C03657=1167.639,225.132,-63.200,-177.659,7.224,148.674
C03658=1167.644,224.883,-63.174,-177.662,7.221,148.674
C03659=1167.648,224.634,-63.149,-177.665,7.219,148.674
C03660=1167.653,224.386,-63.123,-177.668,7.216,148.674
C03661=1167.657,224.138,-63.098,-177.670,7.214,148.674
C03662=1167.661,223.888,-63.073,-177.673,7.212,148.675
C03663=1167.666,223.640,-63.047,-177.676,7.210,148.675
C03664=1167.670,223.391,-63.021,-177.679,7.207,148.675
C03665=1167.675,223.142,-62.996,-177.681,7.205,148.675
C03666=1167.680,222.894,-62.970,-177.684,7.202,148.675
C03667=1167.684,222.645,-62.945,-177.686,7.200,148.676
C03668=1167.689,222.397,-62.920,-177.689,7.197,148.676
C03669=1167.693,222.148,-62.894,-177.692,7.195,148.676
C03670=1167.698,221.899,-62.869,-177.695,7.192,148.676
C03671=1167.702,221.650,-62.844,-177.697,7.191,148.676
C03672=1167.707,221.402,-62.818,-177.700,7.188,148.677
C03673=1167.712,221.153,-62.793,-177.703,7.186,148.677
C03674=1167.715,220.904,-62.768,-177.705,7.183,148.677
C03675=1167.720,220.656,-62.743,-177.708,7.181,148.677
C03676=1167.725,220.407,-62.718,-177.711,7.178,148.677
C03677=1167.729,220.158,-62.692,-177.714,7.176,148.678
C03678=1167.734,219.910,-62.667,-177.716,7.174,148.678
C03679=1167.738,219.661,-62.642,-177.719,7.171,148.678
C03680=1167.742,219.413,-62.617,-177.722,7.169,148.678
C03681=1167.747,219.163,-62.592,-177.724,7.166,148.678
C03682=1167.752,218.915,-62.566,-177.727,7.164,148.679
C03683=1167.756,218.666,-62.541,-177.730,7.161,148.679
C03684=1167.761,218.418,-62.516,-177.733,7.159,148.679
C03685=1167.765,218.169,-62.491,-177.735,7.157,148.679
C03686=1167.770,217.921,-62.466,-177.738,7.155,148.679
C03687=1167.774,217.671,-62.441,-177.740,7.152,148.680
C03688=1167.779,217.423,-62.416,-177.743,7.150,148.680
C03689=1167.783,217.174,-62.391,-177.746,7.148,148.680
C03690=1167.788,216.926,-62.366,-177.749,7.145,148.680
C03691=1167.792,216.676,-62.341,-177.751,7.143,148.680
C03692=1167.797,216.428,-62.315,-177.754,7.140,148.681
C03693=1167.801,216.179,-62.291,-177.757,7.138,148.681
C03694=1167.806,215.931,-62.266,-177.760,7.136,148.681
C03695=1167.810,215.682,-62.241,-177.762,7.134,148.681
C03696=1167.815,215.433,-62.216,-177.765,7.131,148.682
C03697=1167.819,215.184,-62.191,-177.767,7.129,148.682
C03698=1167.824,214.936,-62.166,-177.771,7.126,148.682
C03699=1167.829,214.687,-62.141,-177.773,7.124,148.682
C03700=1167.833,214.438,-62.116,-177.776,7.122,148.682
C03701=1167.838,214.190,-62.092,-177.779,7.120,148.683
C03702=1167.842,213.940,-62.067,-177.781,7.117,148.683
C03703=1167.846,213.693,-62.042,-177.784,7.115,148.683
C03704=1167.851,213.443,-62.017,-177.786,7.113,148.683
C03705=1167.855,213.195,-61.993,-177.790,7.110,148.684
C03706=1167.860,212.946,-61.968,-177.792,7.108,148.684
C03707=1167.865,212.697,-61.942,-177.795,7.106,148.684
C03708=1167.869,212.449,-61.918,-177.797,7.103,148.684
C03709=1167.873,212.199,-61.893,-177.800,7.101,148.685
C03710=1167.878,211.951,-61.869,-177.803,7.099,148.685
C03711=1167.883,211.703,-61.844,-177.806,7.096,148.685
C03712=1167.887,211.453,-61.819,-177.809,7.094,148.685
C03713=1167.892,211.205,-61.795,-177.811,7.092,148.685
C03714=1167.897,210.956,-61.770,-177.814,7.090,148.686
C03715=1167.901,210.707,-61.745,-177.816,7.087,148.686
C03716=1167.906,210.437,-61.719,-177.819,7.085,148.686
C03717=1167.910,210.166,-61.692,-177.823,7.082,148.687
C03718=1167.915,209.896,-61.665,-177.825,7.080,148.687
C03719=1167.921,209.626,-61.638,-177.828,7.078,148.687
C03720=1167.925,209.376,-61.613,-177.831,7.075,148.687
C03721=1167.929,209.128,-61.589,-177.834,7.073,148.687
C03722=1167.935,208.879,-61.564,-177.836,7.071,148.688
C03723=1167.938,208.630,-61.540,-177.839,7.068,148.688
C03724=1167.944,208.381,-61.515,-177.842,7.066,148.688
C03725=1167.948,208.133,-61.491,-177.844,7.063,148.688
C03726=1167.953,207.884,-61.467,-177.847,7.062,148.689
C03727=1167.957,207.635,-61.442,-177.850,7.059,148.689
C03728=1167.961,207.387,-61.418,-177.853,7.057,148.689
C03729=1167.966,207.138,-61.393,-177.855,7.055,148.689
C03730=1167.970,206.889,-61.369,-177.858,7.052,148.689
C03731=1167.975,206.640,-61.344,-177.861,7.050,148.690
C03732=1167.980,206.392,-61.320,-177.864,7.048,148.690
C03733=1167.985,206.143,-61.296,-177.866,7.046,148.690
C03734=1167.989,205.894,-61.271,-177.869,7.044,148.691
C03735=1167.993,205.645,-61.247,-177.872,7.041,148.691
C03736=1167.998,205.397,-61.222,-177.874,7.039,148.691
C03737=1168.003,205.148,-61.199,-177.877,7.036,148.691
C03738=1168.007,204.899,-61.175,-177.880,7.034,148.691
C03739=1168.012,204.650,-61.150,-177.882,7.033,148.692
C03740=1168.016,204.401,-61.126,-177.885,7.030,148.692
C03741=1168.021,204.153,-61.102,-177.888,7.028,148.692
C03742=1168.025,203.904,-61.077,-177.891,7.025,148.693
C03743=1168.030,203.655,-61.053,-177.893,7.023,148.693
C03744=1168.034,203.406,-61.029,-177.896,7.021,148.693
C03745=1168.039,203.157,-61.005,-177.899,7.019,148.693
C03746=1168.044,202.909,-60.981,-177.901,7.017,148.694
C03747=1168.048,202.660,-60.956,-177.904,7.015,148.694
C03748=1168.053,202.411,-60.932,-177.907,7.012,148.694
C03749=1168.057,202.162,-60.908,-177.909,7.010,148.694
C03750=1168.062,201.914,-60.884,-177.913,7.008,148.695
C03751=1168.066,201.665,-60.861,-177.915,7.006,148.695
C03752=1168.071,201.415,-60.836,-177.918,7.004,148.695
C03753=1168.075,201.167,-60.812,-177.920,7.001,148.695
C03754=1168.080,200.918,-60.787,-177.923,6.999,148.696
C03755=1168.084,200.669,-60.764,-177.926,6.997,148.696
C03756=1168.089,200.421,-60.740,-177.928,6.994,148.696
C03757=1168.094,200.172,-60.716,-177.931,6.993,148.696
C03758=1168.098,199.923,-60.692,-177.934,6.991,148.697
C03759=1168.102,199.674,-60.668,-177.937,6.988,148.697
C03760=1168.107,199.425,-60.644,-177.939,6.986,148.697
C03761=1168.112,199.177,-60.620,-177.943,6.983,148.697
C03762=1168.117,198.927,-60.596,-177.945,6.981,148.698
C03763=1168.121,198.679,-60.572,-177.947,6.980,148.698
C03764=1168.126,198.431,-60.548,-177.951,6.977,148.698
C03765=1168.130,198.182,-60.525,-177.953,6.975,148.698
C03766=1168.134,197.932,-60.500,-177.956,6.973,148.699
C03767=1168.139,197.683,-60.477,-177.959,6.971,148.699
C03768=1168.143,197.435,-60.453,-177.961,6.968,148.699
C03769=1168.148,197.186,-60.429,-177.964,6.967,148.700
C03770=1168.153,196.937,-60.405,-177.967,6.964,148.700
C03771=1168.158,196.688,-60.381,-177.969,6.962,148.700
C03772=1168.162,196.440,-60.357,-177.972,6.960,148.700
C03773=1168.167,196.191,-60.334,-177.975,6.958,148.701
C03774=1168.171,195.942,-60.310,-177.977,6.955,148.701
C03775=1168.176,195.693,-60.287,-177.980,6.954,148.701
C03776=1168.181,195.444,-60.263,-177.983,6.951,148.701
C03777=1168.185,195.196,-60.239,-177.985,6.949,148.702
C03778=1168.190,194.947,-60.216,-177.988,6.947,148.702
C03779=1168.195,194.698,-60.192,-177.991,6.945,148.702
C03780=1168.199,194.449,-60.168,-177.993,6.942,148.702
C03781=1168.204,194.200,-60.145,-177.996,6.941,148.703
C03782=1168.207,193.951,-60.120,-177.999,6.939,148.703
C03783=1168.212,193.702,-60.097,-178.002,6.936,148.703
C03784=1168.217,193.453,-60.074,-178.004,6.934,148.704
C03785=1168.222,193.204,-60.050,-178.007,6.932,148.704
C03786=1168.226,192.956,-60.026,-178.010,6.930,148.704
C03787=1168.231,192.707,-60.003,-178.012,6.928,148.704
C03788=1168.235,192.458,-59.980,-178.015,6.926,148.705
C03789=1168.240,192.209,-59.956,-178.018,6.923,148.705
C03790=1168.244,191.960,-59.932,-178.021,6.921,148.705
C03791=1168.250,191.712,-59.909,-178.023,6.919,148.706
C03792=1168.254,191.463,-59.886,-178.026,6.917,148.706
C03793=1168.259,191.214,-59.862,-178.029,6.915,148.706
C03794=1168.264,190.965,-59.838,-178.031,6.913,148.706
C03795=1168.268,190.716,-59.815,-178.034,6.911,148.707
C03796=1168.273,190.467,-59.792,-178.037,6.909,148.707
C03797=1168.277,190.219,-59.769,-178.039,6.907,148.707
C03798=1168.282,189.970,-59.746,-178.042,6.905,148.708
C03799=1168.286,189.721,-59.722,-178.045,6.902,148.708
C03800=1168.291,189.472,-59.698,-178.048,6.900,148.708
C03801=1168.295,189.223,-59.675,-178.050,6.898,148.708
C03802=1168.300,188.974,-59.651,-178.053,6.897,148.709
C03803=1168.305,188.725,-59.628,-178.056,6.894,148.709
C03804=1168.309,188.476,-59.605,-178.059,6.892,148.709
C03805=1168.313,188.227,-59.582,-178.061,6.890,148.710
C03806=1168.319,187.979,-59.559,-178.064,6.888,148.710
C03807=1168.323,187.730,-59.536,-178.067,6.886,148.710
C03808=1168.328,187.481,-59.512,-178.070,6.884,148.711
C03809=1168.333,187.232,-59.489,-178.072,6.882,148.711
C03810=1168.337,186.983,-59.466,-178.075,6.879,148.711
C03811=1168.342,186.734,-59.443,-178.078,6.877,148.711
C03812=1168.346,186.485,-59.419,-178.081,6.876,148.712
C03813=1168.351,186.236,-59.396,-178.083,6.874,148.712
C03814=1168.355,185.987,-59.373,-178.086,6.871,148.712
C03815=1168.360,185.739,-59.350,-178.089,6.869,148.713
C03816=1168.365,185.490,-59.327,-178.091,6.867,148.713
C03817=1168.370,185.241,-59.304,-178.094,6.865,148.713
C03818=1168.374,184.992,-59.281,-178.097,6.863,148.713
C03819=1168.378,184.743,-59.257,-178.100,6.861,148.714
C03820=1168.384,184.473,-59.232,-178.102,6.859,148.714
C03821=1168.388,184.204,-59.208,-178.105,6.857,148.715
C03822=1168.393,183.934,-59.183,-178.108,6.855,148.715
C03823=1168.399,183.664,-59.158,-178.111,6.852,148.715
C03824=1168.403,183.416,-59.135,-178.114,6.850,148.715
C03825=1168.407,183.167,-59.112,-178.116,6.848,148.716
C03826=1168.413,182.918,-59.089,-178.120,6.846,148.716
C03827=1168.417,182.670,-59.066,-178.122,6.844,148.716
C03828=1168.422,182.420,-59.043,-178.125,6.842,148.717
C03829=1168.426,182.171,-59.020,-178.127,6.840,148.717
C03830=1168.430,181.922,-58.997,-178.130,6.838,148.717
C03831=1168.436,181.674,-58.974,-178.133,6.836,148.718
C03832=1168.440,181.425,-58.951,-178.136,6.834,148.718
C03833=1168.445,181.175,-58.929,-178.138,6.832,148.718
C03834=1168.449,180.926,-58.905,-178.141,6.830,148.718
C03835=1168.454,180.678,-58.883,-178.144,6.828,148.719
C03836=1168.459,180.429,-58.860,-178.147,6.826,148.719
C03837=1168.463,180.180,-58.838,-178.149,6.824,148.720
C03838=1168.468,179.931,-58.814,-178.152,6.822,148.720
C03839=1168.472,179.682,-58.793,-178.154,6.820,148.720
C03840=1168.477,179.433,-58.769,-178.157,6.818,148.720
C03841=1168.482,179.184,-58.746,-178.160,6.816,148.721
C03842=1168.486,178.935,-58.724,-178.163,6.814,148.721
C03843=1168.491,178.687,-58.701,-178.165,6.812,148.721
C03844=1168.495,178.438,-58.678,-178.168,6.810,148.722
C03845=1168.500,178.188,-58.655,-178.171,6.808,148.722
C03846=1168.504,177.940,-58.633,-178.174,6.806,148.722
C03847=1168.510,177.691,-58.610,-178.176,6.804,148.723
C03848=1168.514,177.442,-58.588,-178.179,6.802,148.723
C03849=1168.519,177.192,-58.565,-178.182,6.801,148.723
C03850=1168.524,176.944,-58.543,-178.184,6.798,148.723
C03851=1168.527,176.695,-58.520,-178.187,6.796,148.724
C03852=1168.532,176.446,-58.497,-178.190,6.794,148.724
C03853=1168.537,176.198,-58.475,-178.192,6.792,148.725
C03854=1168.542,175.948,-58.452,-178.195,6.791,148.725
C03855=1168.546,175.699,-58.429,-178.198,6.788,148.725
C03856=1168.552,175.450,-58.407,-178.201,6.786,148.725
C03857=1168.556,175.201,-58.385,-178.203,6.784,148.726
C03858=1168.561,174.952,-58.362,-178.206,6.782,148.726
C03859=1168.565,174.703,-58.340,-178.209,6.781,148.727
C03860=1168.569,174.455,-58.317,-178.211,6.779,148.727
C03861=1168.574,174.205,-58.295,-178.215,6.776,148.727
C03862=1168.579,173.957,-58.272,-178.217,6.774,148.727
C03863=1168.583,173.708,-58.250,-178.219,6.772,148.728
C03864=1168.589,173.459,-58.228,-178.222,6.771,148.728
C03865=1168.593,173.210,-58.205,-178.225,6.769,148.728
C03866=1168.598,172.960,-58.182,-178.228,6.767,148.729
C03867=1168.603,172.712,-58.161,-178.231,6.765,148.729
C03868=1168.607,172.463,-58.138,-178.233,6.763,148.730
C03869=1168.612,172.214,-58.116,-178.236,6.761,148.730
C03870=1168.617,171.965,-58.094,-178.238,6.759,148.730
C03871=1168.620,171.716,-58.071,-178.241,6.757,148.730
C03872=1168.625,171.467,-58.049,-178.244,6.755,148.731
C03873=1168.630,171.218,-58.027,-178.247,6.753,148.731
C03874=1168.635,170.970,-58.004,-178.250,6.751,148.731
C03875=1168.639,170.720,-57.982,-178.252,6.749,148.732
C03876=1168.645,170.471,-57.960,-178.255,6.748,148.732
C03877=1168.649,170.222,-57.938,-178.258,6.746,148.733
C03878=1168.653,169.973,-57.916,-178.260,6.744,148.733
C03879=1168.658,169.725,-57.893,-178.263,6.742,148.733
C03880=1168.663,169.475,-57.871,-178.266,6.739,148.733
C03881=1168.668,169.226,-57.849,-178.269,6.738,148.734
C03882=1168.672,168.977,-57.827,-178.271,6.736,148.734
C03883=1168.677,168.728,-57.805,-178.274,6.734,148.735
C03884=1168.682,168.479,-57.782,-178.277,6.732,148.735
C03885=1168.686,168.231,-57.760,-178.279,6.731,148.735
C03886=1168.691,167.981,-57.738,-178.282,6.729,148.736
C03887=1168.696,167.733,-57.717,-178.284,6.727,148.736
C03888=1168.700,167.483,-57.695,-178.288,6.724,148.736
C03889=1168.705,167.235,-57.672,-178.290,6.722,148.737
C03890=1168.710,166.985,-57.650,-178.293,6.721,148.737
C03891=1168.715,166.737,-57.629,-178.296,6.719,148.737
C03892=1168.719,166.487,-57.606,-178.298,6.717,148.738
C03893=1168.724,166.239,-57.585,-178.301,6.715,148.738
C03894=1168.728,165.989,-57.563,-178.304,6.714,148.738
C03895=1168.733,165.741,-57.541,-178.306,6.712,148.739
C03896=1168.738,165.491,-57.518,-178.309,6.710,148.739
C03897=1168.743,165.242,-57.497,-178.312,6.708,148.739
C03898=1168.747,164.993,-57.475,-178.315,6.705,148.740
C03899=1168.752,164.744,-57.453,-178.317,6.704,148.740
C03900=1168.757,164.496,-57.431,-178.320,6.702,148.740
C03901=1168.761,164.246,-57.409,-178.323,6.700,148.741
C03902=1168.766,163.998,-57.388,-178.325,6.698,148.741
C03903=1168.770,163.748,-57.366,-178.328,6.697,148.741
C03904=1168.775,163.500,-57.344,-178.331,6.695,148.742
C03905=1168.779,163.250,-57.322,-178.333,6.693,148.742
C03906=1168.784,163.002,-57.300,-178.336,6.691,148.743
C03907=1168.789,162.753,-57.278,-178.339,6.689,148.743
C03908=1168.793,162.504,-57.256,-178.342,6.687,148.743
C03909=1168.798,162.255,-57.235,-178.345,6.685,148.744
C03910=1168.803,162.005,-57.213,-178.347,6.684,148.744
C03911=1168.808,161.756,-57.192,-178.350,6.682,148.744
C03912=1168.813,161.508,-57.170,-178.353,6.680,148.745
C03913=1168.817,161.259,-57.148,-178.355,6.678,148.745
C03914=1168.822,161.010,-57.126,-178.358,6.676,148.745
C03915=1168.826,160.761,-57.104,-178.360,6.674,148.746
C03916=1168.831,160.511,-57.083,-178.363,6.673,148.746
C03917=1168.836,160.263,-57.062,-178.366,6.671,148.746
C03918=1168.840,160.013,-57.040,-178.368,6.669,148.747
C03919=1168.845,159.765,-57.018,-178.371,6.667,148.747
C03920=1168.850,159.515,-56.997,-178.374,6.665,148.748
C03921=1168.855,159.266,-56.975,-178.377,6.663,148.748
C03922=1168.859,159.017,-56.953,-178.380,6.661,148.748
C03923=1168.864,158.769,-56.931,-178.382,6.660,148.749
C03924=1168.869,158.500,-56.909,-178.385,6.658,148.749
C03925=1168.875,158.230,-56.885,-178.388,6.656,148.749
C03926=1168.879,157.961,-56.863,-178.391,6.654,148.750
C03927=1168.884,157.693,-56.839,-178.394,6.652,148.750
C03928=1168.890,157.443,-56.818,-178.397,6.650,148.751
C03929=1168.893,157.194,-56.796,-178.399,6.648,148.751
C03930=1168.898,156.946,-56.774,-178.402,6.647,148.751
C03931=1168.903,156.696,-56.753,-178.405,6.645,148.752
C03932=1168.907,156.447,-56.731,-178.407,6.643,148.752
C03933=1168.913,156.198,-56.710,-178.410,6.641,148.752
C03934=1168.917,155.949,-56.689,-178.413,6.640,148.753
C03935=1168.922,155.701,-56.667,-178.415,6.638,148.753
C03936=1168.926,155.451,-56.646,-178.418,6.636,148.754
C03937=1168.931,155.202,-56.625,-178.421,6.634,148.754
C03938=1168.936,154.953,-56.604,-178.423,6.633,148.754
C03939=1168.941,154.704,-56.582,-178.426,6.631,148.755
C03940=1168.946,154.454,-56.561,-178.429,6.629,148.755
C03941=1168.950,154.206,-56.540,-178.432,6.627,148.755
C03942=1168.955,153.957,-56.519,-178.434,6.626,148.756
C03943=1168.960,153.708,-56.497,-178.437,6.624,148.756
C03944=1168.964,153.458,-56.476,-178.440,6.621,148.757
C03945=1168.969,153.210,-56.455,-178.443,6.620,148.757
C03946=1168.974,152.961,-56.434,-178.446,6.618,148.757
C03947=1168.979,152.712,-56.412,-178.448,6.616,148.758
C03948=1168.984,152.463,-56.391,-178.451,6.614,148.758
C03949=1168.988,152.213,-56.370,-178.454,6.613,148.758
C03950=1168.992,151.964,-56.348,-178.456,6.611,148.759
C03951=1168.998,151.715,-56.328,-178.459,6.609,148.759
C03952=1169.002,151.467,-56.306,-178.462,6.607,148.760
C03953=1169.007,151.218,-56.285,-178.464,6.606,148.760
C03954=1169.012,150.968,-56.264,-178.467,6.604,148.760
C03955=1169.016,150.719,-56.243,-178.470,6.602,148.761
C03956=1169.021,150.470,-56.222,-178.473,6.601,148.761
C03957=1169.026,150.221,-56.201,-178.476,6.599,148.762
C03958=1169.030,149.972,-56.180,-178.478,6.597,148.762
C03959=1169.035,149.723,-56.159,-178.481,6.595,148.762
C03960=1169.040,149.473,-56.138,-178.484,6.594,148.763
C03961=1169.044,149.225,-56.117,-178.486,6.592,148.763
C03962=1169.049,148.976,-56.096,-178.489,6.590,148.764
C03963=1169.054,148.726,-56.075,-178.492,6.588,148.764
C03964=1169.059,148.477,-56.054,-178.495,6.587,148.764
C03965=1169.064,148.229,-56.033,-178.497,6.585,148.765
C03966=1169.068,147.980,-56.012,-178.500,6.583,148.765
C03967=1169.073,147.731,-55.991,-178.503,6.581,148.766
C03968=1169.077,147.481,-55.971,-178.505,6.580,148.766
C03969=1169.082,147.232,-55.950,-178.507,6.579,148.766
C03970=1169.087,146.983,-55.928,-178.510,6.577,148.767
C03971=1169.092,146.734,-55.908,-178.513,6.575,148.767
C03972=1169.097,146.485,-55.887,-178.516,6.574,148.767
C03973=1169.101,146.236,-55.866,-178.518,6.572,148.768
C03974=1169.106,145.987,-55.845,-178.521,6.570,148.768
C03975=1169.111,145.738,-55.825,-178.524,6.568,148.769
C03976=1169.116,145.488,-55.804,-178.526,6.567,148.769
C03977=1169.120,145.240,-55.783,-178.529,6.565,148.769
C03978=1169.125,144.991,-55.762,-178.532,6.563,148.770
C03979=1169.129,144.741,-55.741,-178.535,6.562,148.770
C03980=1169.134,144.492,-55.720,-178.538,6.560,148.771
C03981=1169.139,144.243,-55.700,-178.540,6.558,148.771
C03982=1169.144,143.994,-55.679,-178.543,6.556,148.772
C03983=1169.148,143.745,-55.658,-178.546,6.555,148.772
C03984=1169.154,143.495,-55.637,-178.548,6.553,148.772
C03985=1169.158,143.246,-55.617,-178.551,6.551,148.773
C03986=1169.162,142.998,-55.597,-178.554,6.550,148.773
C03987=1169.168,142.748,-55.576,-178.557,6.548,148.773
C03988=1169.172,142.499,-55.555,-178.559,6.546,148.774
C03989=1169.177,142.250,-55.534,-178.562,6.544,148.774
C03990=1169.182,142.001,-55.514,-178.565,6.543,148.775
C03991=1169.187,141.752,-55.493,-178.567,6.541,148.775
C03992=1169.191,141.503,-55.473,-178.569,6.540,148.775
C03993=1169.196,141.254,-55.452,-178.573,6.538,148.776
C03994=1169.201,141.005,-55.431,-178.575,6.537,148.776
C03995=1169.205,140.756,-55.411,-178.578,6.535,148.777
C03996=1169.210,140.507,-55.391,-178.581,6.533,148.777
C03997=1169.215,140.257,-55.370,-178.583,6.532,148.778
C03998=1169.220,140.008,-55.350,-178.586,6.530,148.778
C03999=1169.224,139.759,-55.330,-178.589,6.528,148.778
C04000=1169.229,139.510,-55.309,-178.592,6.526,148.779
C04001=1169.234,139.261,-55.288,-178.594,6.525,148.779
C04002=1169.238,139.012,-55.268,-178.597,6.523,148.779
C04003=1169.243,138.763,-55.247,-178.600,6.521,148.780
C04004=1169.248,138.513,-55.227,-178.603,6.520,148.780
C04005=1169.253,138.264,-55.207,-178.605,6.519,148.781
C04006=1169.258,138.015,-55.186,-178.608,6.517,148.781
C04007=1169.263,137.767,-55.166,-178.610,6.515,148.782
C04008=1169.267,137.518,-55.146,-178.613,6.514,148.782
C04009=1169.272,137.268,-55.126,-178.616,6.512,148.782
C04010=1169.277,137.019,-55.105,-178.618,6.510,148.783
C04011=1169.282,136.770,-55.085,-178.621,6.508,148.783
C04012=1169.286,136.520,-55.065,-178.624,6.507,148.784
C04013=1169.291,136.271,-55.045,-178.627,6.505,148.784
C04014=1169.296,136.022,-55.024,-178.630,6.504,148.785
C04015=1169.300,135.773,-55.003,-178.632,6.502,148.785
C04016=1169.305,135.524,-54.984,-178.635,6.501,148.785
C04017=1169.309,135.275,-54.963,-178.637,6.499,148.786
C04018=1169.315,135.026,-54.943,-178.640,6.497,148.786
C04019=1169.320,134.776,-54.923,-178.643,6.496,148.787
C04020=1169.324,134.528,-54.903,-178.645,6.494,148.787
C04021=1169.329,134.279,-54.882,-178.649,6.493,148.788
C04022=1169.334,134.029,-54.863,-178.651,6.491,148.788
C04023=1169.338,133.780,-54.842,-178.654,6.489,148.788
C04024=1169.344,133.530,-54.822,-178.657,6.487,148.789
C04025=1169.349,133.282,-54.802,-178.659,6.486,148.789
C04026=1169.353,133.033,-54.782,-178.661,6.485,148.790
C04027=1169.358,132.783,-54.762,-178.664,6.483,148.790
C04028=1169.363,132.514,-54.740,-178.667,6.482,148.791
C04029=1169.368,132.246,-54.718,-178.670,6.480,148.791
C04030=1169.373,131.978,-54.697,-178.673,6.478,148.791
C04031=1169.379,131.709,-54.676,-178.677,6.476,148.792
C04032=1169.383,131.460,-54.655,-178.679,6.475,148.792
C04033=1169.388,131.210,-54.636,-178.681,6.473,148.793
C04034=1169.392,130.961,-54.615,-178.684,6.472,148.793
C04035=1169.398,130.712,-54.596,-178.687,6.470,148.793
C04036=1169.402,130.464,-54.576,-178.689,6.468,148.794
C04037=1169.407,130.214,-54.556,-178.693,6.467,148.794
C04038=1169.412,129.965,-54.535,-178.695,6.465,148.795
C04039=1169.417,129.716,-54.516,-178.698,6.464,148.795
C04040=1169.422,129.467,-54.495,-178.700,6.462,148.796
C04041=1169.426,129.217,-54.476,-178.703,6.461,148.796
C04042=1169.431,128.968,-54.456,-178.706,6.459,148.796
C04043=1169.436,128.720,-54.436,-178.709,6.457,148.797
C04044=1169.441,128.470,-54.416,-178.712,6.456,148.797
C04045=1169.445,128.221,-54.396,-178.714,6.455,148.798
C04046=1169.450,127.971,-54.376,-178.716,6.453,148.798
C04047=1169.455,127.722,-54.357,-178.719,6.451,148.799
C04048=1169.460,127.474,-54.337,-178.722,6.450,148.799
C04049=1169.465,127.224,-54.317,-178.725,6.448,148.800
C04050=1169.469,126.974,-54.297,-178.728,6.446,148.800
C04051=1169.474,126.726,-54.277,-178.730,6.445,148.800
C04052=1169.478,126.477,-54.258,-178.732,6.444,148.801
C04053=1169.483,126.227,-54.239,-178.735,6.442,148.801
C04054=1169.488,125.978,-54.219,-178.738,6.440,148.802
C04055=1169.493,125.730,-54.199,-178.741,6.439,148.802
C04056=1169.498,125.480,-54.179,-178.744,6.437,148.803
C04057=1169.502,125.230,-54.160,-178.746,6.436,148.803
C04058=1169.508,124.982,-54.140,-178.749,6.435,148.804
C04059=1169.512,124.733,-54.120,-178.751,6.433,148.804
C04060=1169.517,124.483,-54.100,-178.755,6.432,148.805
C04061=1169.522,124.234,-54.081,-178.757,6.430,148.805
C04062=1169.527,123.985,-54.061,-178.760,6.428,148.805
C04063=1169.531,123.735,-54.042,-178.762,6.427,148.806
C04064=1169.536,123.487,-54.022,-178.765,6.425,148.806
C04065=1169.541,123.238,-54.003,-178.768,6.424,148.807
C04066=1169.546,122.988,-53.983,-178.771,6.422,148.807
C04067=1169.551,122.739,-53.964,-178.773,6.421,148.808
C04068=1169.556,122.490,-53.944,-178.776,6.420,148.808
C04069=1169.560,122.240,-53.924,-178.778,6.418,148.808
C04070=1169.565,121.991,-53.906,-178.781,6.417,148.809
C04071=1169.569,121.742,-53.885,-178.784,6.415,148.809
C04072=1169.574,121.493,-53.866,-178.787,6.413,148.810
C04073=1169.580,121.244,-53.846,-178.789,6.412,148.810
C04074=1169.584,120.994,-53.827,-178.792,6.410,148.811
C04075=1169.589,120.746,-53.808,-178.795,6.409,148.811
C04076=1169.594,120.496,-53.788,-178.798,6.407,148.812
C04077=1169.598,120.247,-53.769,-178.800,6.406,148.812
C04078=1169.604,119.998,-53.749,-178.802,6.405,148.812
C04079=1169.608,119.749,-53.730,-178.806,6.403,148.813
C04080=1169.613,119.500,-53.711,-178.808,6.402,148.813
C04081=1169.618,119.250,-53.691,-178.811,6.400,148.814
C04082=1169.623,119.001,-53.672,-178.813,6.399,148.814
C04083=1169.627,118.752,-53.653,-178.816,6.397,148.815
C04084=1169.632,118.503,-53.633,-178.819,6.396,148.815
C04085=1169.637,118.254,-53.614,-178.822,6.394,148.816
C04086=1169.642,118.004,-53.594,-178.824,6.392,148.816
C04087=1169.647,117.756,-53.576,-178.827,6.392,148.816
C04088=1169.652,117.505,-53.557,-178.830,6.390,148.817
C04089=1169.656,117.256,-53.537,-178.833,6.388,148.818
C04090=1169.661,117.007,-53.518,-178.835,6.387,148.818
C04091=1169.666,116.758,-53.499,-178.837,6.386,148.818
C04092=1169.671,116.509,-53.479,-178.841,6.384,148.819
C04093=1169.675,116.260,-53.460,-178.843,6.383,148.819
C04094=1169.680,116.011,-53.441,-178.846,6.381,148.820
C04095=1169.685,115.761,-53.421,-178.848,6.380,148.820
C04096=1169.690,115.512,-53.403,-178.851,6.378,148.821
C04097=1169.695,115.262,-53.384,-178.854,6.377,148.821
C04098=1169.700,115.013,-53.365,-178.857,6.375,148.822
C04099=1169.704,114.764,-53.345,-178.859,6.374,148.822
C04100=1169.710,114.515,-53.326,-178.862,6.373,148.822
C04101=1169.714,114.265,-53.308,-178.865,6.371,148.823
C04102=1169.719,114.017,-53.289,-178.867,6.370,148.823
C04103=1169.724,113.767,-53.269,-178.870,6.369,148.824
C04104=1169.729,113.519,-53.250,-178.872,6.367,148.824
C04105=1169.734,113.268,-53.231,-178.875,6.366,148.825
C04106=1169.738,113.020,-53.213,-178.878,6.364,148.825
C04107=1169.743,112.770,-53.193,-178.880,6.363,148.826
C04108=1169.748,112.522,-53.174,-178.884,6.362,148.826
C04109=1169.753,112.272,-53.156,-178.886,6.360,148.827
C04110=1169.758,112.023,-53.136,-178.889,6.358,148.827
C04111=1169.763,111.774,-53.117,-178.891,6.357,148.828
C04112=1169.768,111.524,-53.098,-178.894,6.356,148.828
C04113=1169.772,111.275,-53.080,-178.897,6.354,148.829
C04114=1169.777,111.026,-53.060,-178.899,6.353,148.829
C04115=1169.782,110.777,-53.042,-178.902,6.352,148.829
C04116=1169.787,110.527,-53.022,-178.905,6.350,148.830
C04117=1169.792,110.278,-53.004,-178.908,6.348,148.830
C04118=1169.797,110.029,-52.985,-178.910,6.348,148.831
C04119=1169.801,109.780,-52.966,-178.913,6.346,148.831
C04120=1169.807,109.530,-52.947,-178.916,6.344,148.832
C04121=1169.811,109.281,-52.928,-178.918,6.344,148.832
C04122=1169.815,109.032,-52.910,-178.921,6.342,148.833
C04123=1169.821,108.783,-52.891,-178.924,6.340,148.833
C04124=1169.825,108.534,-52.872,-178.927,6.339,148.834
C04125=1169.830,108.284,-52.853,-178.929,6.338,148.834
C04126=1169.834,108.035,-52.834,-178.931,6.336,148.835
C04127=1169.840,107.785,-52.816,-178.935,6.335,148.835
C04128=1169.845,107.537,-52.797,-178.937,6.334,148.836
C04129=1169.849,107.287,-52.779,-178.939,6.332,148.836
C04130=1169.854,107.038,-52.760,-178.943,6.331,148.837
C04131=1169.859,106.789,-52.742,-178.945,6.329,148.837
C04132=1169.864,106.520,-52.721,-178.948,6.328,148.838
C04133=1169.869,106.252,-52.701,-178.951,6.327,148.838
C04134=1169.875,105.983,-52.681,-178.953,6.325,148.839
C04135=1169.880,105.715,-52.662,-178.957,6.324,148.839
C04136=1169.885,105.466,-52.642,-178.959,6.322,148.840
C04137=1169.890,105.216,-52.624,-178.961,6.321,148.840
C04138=1169.894,104.968,-52.605,-178.965,6.320,148.841
C04139=1169.899,104.718,-52.586,-178.967,6.318,148.841
C04140=1169.904,104.469,-52.568,-178.970,6.316,148.841
C04141=1169.909,104.220,-52.550,-178.973,6.316,148.842
C04142=1169.914,103.970,-52.531,-178.975,6.314,148.843
C04143=1169.919,103.721,-52.513,-178.978,6.312,148.843
C04144=1169.924,103.472,-52.494,-178.981,6.312,148.844
C04145=1169.929,103.222,-52.475,-178.983,6.310,148.844
C04146=1169.934,102.973,-52.457,-178.986,6.308,148.844
C04147=1169.938,102.724,-52.438,-178.988,6.308,148.845
C04148=1169.943,102.475,-52.420,-178.992,6.306,148.845
C04149=1169.948,102.225,-52.402,-178.994,6.304,148.846
C04150=1169.953,101.976,-52.383,-178.996,6.304,148.846
C04151=1169.958,101.727,-52.365,-179.000,6.302,148.847
C04152=1169.963,101.478,-52.347,-179.002,6.300,148.847
C04153=1169.968,101.228,-52.328,-179.004,6.300,148.848
C04154=1169.972,100.979,-52.309,-179.008,6.298,148.848
C04155=1169.977,100.730,-52.291,-179.010,6.297,148.849
C04156=1169.982,100.481,-52.273,-179.013,6.296,148.849
C04157=1169.986,100.231,-52.255,-179.016,6.294,148.850
C04158=1169.992,99.981,-52.236,-179.018,6.293,148.850
C04159=1169.997,99.733,-52.218,-179.021,6.292,148.851
C04160=1170.001,99.484,-52.200,-179.024,6.290,148.851
C04161=1170.006,99.234,-52.181,-179.026,6.289,148.852
C04162=1170.011,98.985,-52.163,-179.029,6.288,148.852
C04163=1170.016,98.735,-52.145,-179.032,6.286,148.853
C04164=1170.021,98.486,-52.127,-179.034,6.285,148.853
C04165=1170.026,98.237,-52.109,-179.037,6.284,148.854
C04166=1170.030,97.988,-52.090,-179.040,6.282,148.854
C04167=1170.035,97.738,-52.072,-179.042,6.281,148.855
C04168=1170.040,97.489,-52.054,-179.045,6.280,148.855
C04169=1170.045,97.240,-52.036,-179.047,6.279,148.856
C04170=1170.050,96.991,-52.018,-179.050,6.278,148.856
C04171=1170.055,96.741,-51.999,-179.053,6.276,148.857
C04172=1170.060,96.491,-51.981,-179.055,6.275,148.857
C04173=1170.065,96.242,-51.963,-179.058,6.274,148.858
C04174=1170.070,95.993,-51.945,-179.061,6.272,148.858
C04175=1170.075,95.744,-51.927,-179.063,6.271,148.859
C04176=1170.079,95.495,-51.909,-179.066,6.270,148.859
C04177=1170.084,95.246,-51.891,-179.068,6.269,148.860
C04178=1170.089,94.996,-51.873,-179.072,6.267,148.860
C04179=1170.094,94.747,-51.855,-179.074,6.266,148.861
C04180=1170.098,94.497,-51.837,-179.077,6.265,148.861
C04181=1170.103,94.248,-51.819,-179.080,6.263,148.862
C04182=1170.108,93.999,-51.801,-179.082,6.262,148.862
C04183=1170.113,93.750,-51.783,-179.085,6.261,148.863
C04184=1170.118,93.501,-51.765,-179.088,6.259,148.863
C04185=1170.123,93.251,-51.747,-179.090,6.259,148.864
C04186=1170.127,93.002,-51.728,-179.093,6.257,148.864
C04187=1170.132,92.752,-51.710,-179.095,6.256,148.865
C04188=1170.137,92.503,-51.693,-179.098,6.255,148.865
C04189=1170.142,92.253,-51.675,-179.101,6.253,148.866
C04190=1170.147,92.004,-51.657,-179.103,6.252,148.866
C04191=1170.152,91.755,-51.639,-179.106,6.251,148.867
C04192=1170.157,91.506,-51.621,-179.109,6.250,148.867
C04193=1170.162,91.257,-51.603,-179.111,6.248,148.868
C04194=1170.167,91.008,-51.585,-179.115,6.247,148.868
C04195=1170.172,90.758,-51.568,-179.117,6.246,148.869
C04196=1170.177,90.509,-51.550,-179.119,6.244,148.869
C04197=1170.182,90.259,-51.532,-179.122,6.244,148.870
C04198=1170.186,90.010,-51.514,-179.125,6.242,148.870
C04199=1170.191,89.760,-51.496,-179.127,6.241,148.871
C04200=1170.196,89.511,-51.479,-179.130,6.240,148.871
C04201=1170.201,89.261,-51.461,-179.133,6.238,148.872
C04202=1170.206,89.013,-51.443,-179.135,6.238,148.872
C04203=1170.210,88.763,-51.425,-179.138,6.236,148.873
C04204=1170.216,88.514,-51.408,-179.140,6.235,148.873
C04205=1170.221,88.264,-51.390,-179.143,6.234,148.874
C04206=1170.225,88.015,-51.372,-179.146,6.232,148.874
C04207=1170.230,87.766,-51.354,-179.149,6.232,148.875
C04208=1170.236,87.516,-51.337,-179.152,6.230,148.875
C04209=1170.241,87.267,-51.319,-179.154,6.229,148.876
C04210=1170.245,87.018,-51.301,-179.157,6.228,148.876
C04211=1170.250,86.768,-51.284,-179.159,6.227,148.877
C04212=1170.255,86.519,-51.266,-179.162,6.225,148.877
C04213=1170.260,86.270,-51.248,-179.164,6.225,148.878
C04214=1170.265,86.020,-51.231,-179.167,6.223,148.878
C04215=1170.269,85.771,-51.213,-179.170,6.221,148.879
C04216=1170.274,85.522,-51.196,-179.172,6.221,148.879
C04217=1170.279,85.272,-51.178,-179.175,6.219,148.880
C04218=1170.284,85.023,-51.160,-179.178,6.218,148.880
C04219=1170.289,84.773,-51.143,-179.181,6.217,148.881
C04220=1170.294,84.525,-51.126,-179.183,6.216,148.881
C04221=1170.299,84.275,-51.108,-179.186,6.214,148.882
C04222=1170.304,84.026,-51.091,-179.189,6.214,148.883
C04223=1170.310,83.777,-51.073,-179.191,6.212,148.883
C04224=1170.314,83.528,-51.056,-179.194,6.210,148.883
C04225=1170.319,83.278,-51.039,-179.197,6.210,148.884
C04226=1170.324,83.029,-51.021,-179.199,6.208,148.884
C04227=1170.329,82.780,-51.003,-179.202,6.208,148.885
C04228=1170.333,82.530,-50.986,-179.205,6.206,148.886
C04229=1170.338,82.280,-50.969,-179.207,6.205,148.886
C04230=1170.343,82.031,-50.951,-179.210,6.204,148.887
C04231=1170.348,81.782,-50.934,-179.212,6.203,148.887
C04232=1170.353,81.532,-50.916,-179.215,6.202,148.888
C04233=1170.358,81.283,-50.899,-179.218,6.201,148.888
C04234=1170.363,81.034,-50.881,-179.220,6.199,148.889
C04235=1170.368,80.785,-50.865,-179.223,6.198,148.889
C04236=1170.373,80.516,-50.846,-179.226,6.197,148.890
C04237=1170.378,80.248,-50.827,-179.229,6.195,148.890
C04238=1170.384,79.980,-50.809,-179.231,6.195,148.891
C04239=1170.389,79.711,-50.790,-179.234,6.193,148.891
C04240=1170.394,79.462,-50.772,-179.237,6.192,148.892
C04241=1170.398,79.212,-50.756,-179.240,6.191,148.892
C04242=1170.404,78.962,-50.738,-179.243,6.190,148.893
C04243=1170.409,78.713,-50.720,-179.245,6.189,148.893
C04244=1170.414,78.464,-50.704,-179.248,6.187,148.894
C04245=1170.419,78.215,-50.687,-179.250,6.187,148.895
C04246=1170.423,77.966,-50.669,-179.253,6.185,148.895
C04247=1170.428,77.716,-50.652,-179.256,6.184,148.896
C04248=1170.433,77.466,-50.635,-179.258,6.183,148.896
C04249=1170.438,77.217,-50.617,-179.261,6.182,148.897
C04250=1170.443,76.968,-50.601,-179.264,6.180,148.897
C04251=1170.448,76.719,-50.584,-179.266,6.180,148.898
C04252=1170.453,76.469,-50.567,-179.269,6.178,148.898
C04253=1170.457,76.220,-50.549,-179.271,6.177,148.899
C04254=1170.463,75.970,-50.532,-179.274,6.176,148.899
C04255=1170.468,75.721,-50.516,-179.277,6.175,148.900
C04256=1170.473,75.472,-50.498,-179.280,6.174,148.900
C04257=1170.477,75.223,-50.481,-179.282,6.173,148.901
C04258=1170.482,74.973,-50.464,-179.285,6.172,148.901
C04259=1170.487,74.723,-50.447,-179.287,6.171,148.902
C04260=1170.493,74.474,-50.430,-179.290,6.169,148.902
C04261=1170.498,74.225,-50.413,-179.293,6.168,148.903
C04262=1170.502,73.975,-50.396,-179.295,6.168,148.903
C04263=1170.506,73.726,-50.379,-179.298,6.166,148.904
C04264=1170.512,73.477,-50.362,-179.300,6.165,148.905
C04265=1170.517,73.228,-50.345,-179.303,6.164,148.905
C04266=1170.522,72.978,-50.328,-179.305,6.163,148.906
C04267=1170.526,72.728,-50.311,-179.309,6.162,148.906
C04268=1170.532,72.479,-50.294,-179.311,6.161,148.907
C04269=1170.537,72.230,-50.278,-179.314,6.159,148.907
C04270=1170.542,71.980,-50.261,-179.316,6.159,148.908
C04271=1170.546,71.731,-50.243,-179.319,6.157,148.908
C04272=1170.551,71.482,-50.227,-179.322,6.157,148.909
C04273=1170.556,71.233,-50.210,-179.324,6.155,148.909
C04274=1170.561,70.983,-50.193,-179.327,6.154,148.910
C04275=1170.566,70.733,-50.176,-179.330,6.153,148.910
C04276=1170.571,70.485,-50.159,-179.332,6.152,148.911
C04277=1170.576,70.235,-50.143,-179.334,6.151,148.911
C04278=1170.581,69.985,-50.125,-179.338,6.150,148.912
C04279=1170.586,69.736,-50.109,-179.340,6.149,148.913
C04280=1170.591,69.487,-50.092,-179.343,6.148,148.913
C04281=1170.596,69.237,-50.075,-179.345,6.147,148.914
C04282=1170.601,68.988,-50.059,-179.348,6.145,148.914
C04283=1170.606,68.739,-50.042,-179.351,6.145,148.915
C04284=1170.610,68.489,-50.025,-179.353,6.143,148.915
C04285=1170.616,68.240,-50.009,-179.356,6.142,148.916
C04286=1170.621,67.991,-49.991,-179.358,6.142,148.916
C04287=1170.626,67.740,-49.975,-179.361,6.140,148.917
C04288=1170.631,67.492,-49.959,-179.363,6.139,148.917
C04289=1170.636,67.242,-49.942,-179.367,6.138,148.918
C04290=1170.640,66.992,-49.925,-179.369,6.137,148.918
C04291=1170.645,66.744,-49.909,-179.372,6.136,148.919
C04292=1170.650,66.494,-49.892,-179.374,6.135,148.920
C04293=1170.655,66.244,-49.875,-179.377,6.134,148.920
C04294=1170.660,65.996,-49.859,-179.380,6.133,148.921
C04295=1170.665,65.745,-49.843,-179.382,6.132,148.921
C04296=1170.669,65.496,-49.826,-179.385,6.131,148.922
C04297=1170.675,65.247,-49.809,-179.388,6.130,148.922
C04298=1170.680,64.997,-49.792,-179.390,6.128,148.923
C04299=1170.685,64.749,-49.776,-179.393,6.128,148.923
C04300=1170.689,64.499,-49.759,-179.395,6.127,148.924
C04301=1170.695,64.249,-49.743,-179.398,6.126,148.925
C04302=1170.700,64.000,-49.727,-179.400,6.125,148.925
C04303=1170.704,63.750,-49.710,-179.404,6.123,148.926
C04304=1170.709,63.502,-49.694,-179.406,6.123,148.926
C04305=1170.715,63.251,-49.677,-179.408,6.122,148.927
C04306=1170.719,63.002,-49.660,-179.411,6.120,148.927
C04307=1170.725,62.753,-49.644,-179.413,6.119,148.928
C04308=1170.729,62.503,-49.627,-179.417,6.118,148.928
C04309=1170.734,62.254,-49.612,-179.419,6.117,148.929
C04310=1170.739,62.005,-49.595,-179.421,6.117,148.929
C04311=1170.745,61.756,-49.578,-179.424,6.115,148.930
C04312=1170.749,61.505,-49.562,-179.427,6.115,148.930
C04313=1170.755,61.257,-49.546,-179.429,6.113,148.931
C04314=1170.759,61.007,-49.529,-179.432,6.112,148.932
C04315=1170.764,60.757,-49.513,-179.434,6.111,148.932
C04316=1170.769,60.508,-49.497,-179.437,6.110,148.933
C04317=1170.773,60.259,-49.480,-179.440,6.109,148.933
C04318=1170.780,60.009,-49.464,-179.443,6.108,148.934
C04319=1170.784,59.760,-49.448,-179.445,6.107,148.934
C04320=1170.789,59.511,-49.431,-179.448,6.107,148.935
C04321=1170.794,59.261,-49.415,-179.450,6.105,148.935
C04322=1170.799,59.012,-49.399,-179.453,6.104,148.936
C04323=1170.804,58.762,-49.383,-179.455,6.104,148.936
C04324=1170.809,58.513,-49.367,-179.458,6.102,148.937
C04325=1170.813,58.264,-49.350,-179.460,6.101,148.938
C04326=1170.819,58.014,-49.335,-179.464,6.100,148.938
C04327=1170.823,57.765,-49.318,-179.466,6.099,148.939
C04328=1170.829,57.515,-49.302,-179.468,6.099,148.939
C04329=1170.833,57.266,-49.286,-179.471,6.097,148.940
C04330=1170.838,57.016,-49.270,-179.474,6.096,148.940
C04331=1170.843,56.767,-49.253,-179.476,6.096,148.941
C04332=1170.849,56.517,-49.237,-179.479,6.094,148.941
C04333=1170.854,56.268,-49.221,-179.482,6.094,148.942
C04334=1170.859,56.018,-49.205,-179.484,6.093,148.943
C04335=1170.864,55.769,-49.189,-179.487,6.092,148.943
C04336=1170.869,55.519,-49.173,-179.489,6.091,148.944
C04337=1170.874,55.271,-49.156,-179.493,6.089,148.944
C04338=1170.879,55.020,-49.140,-179.495,6.089,148.945
C04339=1170.884,54.771,-49.125,-179.497,6.088,148.945
C04340=1170.889,54.503,-49.107,-179.500,6.086,148.946
C04341=1170.894,54.234,-49.090,-179.503,6.086,148.947
C04342=1170.900,53.966,-49.073,-179.506,6.085,148.947
C04343=1170.905,53.697,-49.056,-179.508,6.084,148.948
C04344=1170.910,53.447,-49.040,-179.511,6.082,148.948
C04345=1170.915,53.198,-49.023,-179.514,6.082,148.949
C04346=1170.920,52.949,-49.008,-179.516,6.081,148.949
C04347=1170.924,52.700,-48.992,-179.519,6.080,148.950
C04348=1170.930,52.450,-48.976,-179.522,6.079,148.951
C04349=1170.935,52.200,-48.960,-179.524,6.078,148.951
C04350=1170.940,51.951,-48.944,-179.527,6.077,148.952
C04351=1170.945,51.702,-48.928,-179.530,6.076,148.952
C04352=1170.950,51.452,-48.912,-179.532,6.075,148.953
C04353=1170.955,51.202,-48.897,-179.535,6.074,148.953
C04354=1170.960,50.953,-48.880,-179.537,6.073,148.954
C04355=1170.965,50.704,-48.865,-179.540,6.073,148.955
C04356=1170.970,50.454,-48.850,-179.542,6.071,148.955
C04357=1170.974,50.205,-48.833,-179.545,6.070,148.956
C04358=1170.980,49.956,-48.817,-179.547,6.070,148.956
C04359=1170.985,49.706,-48.802,-179.550,6.068,148.957
C04360=1170.990,49.456,-48.786,-179.553,6.067,148.957
C04361=1170.995,49.207,-48.769,-179.555,6.067,148.958
C04362=1170.999,48.958,-48.754,-179.559,6.066,148.959
C04363=1171.004,48.708,-48.738,-179.561,6.065,148.959
C04364=1171.010,48.459,-48.723,-179.563,6.064,148.960
C04365=1171.015,48.209,-48.707,-179.566,6.062,148.960
C04366=1171.019,47.960,-48.691,-179.569,6.062,148.961
C04367=1171.025,47.710,-48.675,-179.571,6.061,148.961
C04368=1171.030,47.461,-48.660,-179.573,6.061,148.962
C04369=1171.034,47.211,-48.644,-179.576,6.059,148.962
C04370=1171.040,46.962,-48.629,-179.579,6.058,148.963
C04371=1171.045,46.712,-48.613,-179.581,6.058,148.963
C04372=1171.049,46.463,-48.598,-179.584,6.056,148.964
C04373=1171.054,46.214,-48.581,-179.586,6.055,148.965
C04374=1171.060,45.964,-48.566,-179.589,6.055,148.965
C04375=1171.065,45.715,-48.550,-179.592,6.054,148.966
C04376=1171.069,45.465,-48.535,-179.594,6.053,148.966
C04377=1171.074,45.216,-48.519,-179.597,6.052,148.967
C04378=1171.080,44.966,-48.504,-179.599,6.051,148.967
C04379=1171.085,44.716,-48.488,-179.602,6.050,148.968
C04380=1171.089,44.467,-48.473,-179.605,6.049,148.969
C04381=1171.095,44.218,-48.457,-179.607,6.049,148.969
C04382=1171.100,43.968,-48.441,-179.610,6.047,148.970
C04383=1171.104,43.719,-48.426,-179.613,6.047,148.970
C04384=1171.109,43.469,-48.410,-179.615,6.046,148.971
C04385=1171.115,43.220,-48.395,-179.617,6.045,148.971
C04386=1171.119,42.971,-48.380,-179.621,6.044,148.972
C04387=1171.124,42.721,-48.364,-179.623,6.043,148.973
C04388=1171.130,42.471,-48.348,-179.625,6.043,148.973
C04389=1171.134,42.222,-48.333,-179.628,6.041,148.974
C04390=1171.140,41.973,-48.318,-179.631,6.040,148.974
C04391=1171.145,41.723,-48.302,-179.633,6.039,148.975
C04392=1171.149,41.474,-48.287,-179.636,6.039,148.975
C04393=1171.154,41.224,-48.271,-179.638,6.037,148.976
C04394=1171.160,40.975,-48.256,-179.641,6.037,148.977
C04395=1171.165,40.726,-48.241,-179.644,6.036,148.977
C04396=1171.170,40.476,-48.225,-179.646,6.035,148.978
C04397=1171.175,40.226,-48.209,-179.649,6.034,148.978
C04398=1171.179,39.977,-48.194,-179.651,6.033,148.979
C04399=1171.185,39.727,-48.179,-179.654,6.033,148.980
C04400=1171.190,39.478,-48.164,-179.657,6.031,148.980
C04401=1171.195,39.229,-48.149,-179.659,6.031,148.981
C04402=1171.199,38.979,-48.133,-179.662,6.030,148.981
C04403=1171.205,38.729,-48.118,-179.664,6.029,148.982
C04404=1171.210,38.480,-48.102,-179.667,6.028,148.982
C04405=1171.215,38.231,-48.087,-179.669,6.027,148.983
C04406=1171.220,37.981,-48.072,-179.672,6.027,148.984
C04407=1171.225,37.732,-48.057,-179.674,6.026,148.984
C04408=1171.230,37.482,-48.042,-179.677,6.025,148.985
C04409=1171.234,37.233,-48.026,-179.680,6.024,148.985
C04410=1171.240,36.983,-48.011,-179.682,6.023,148.986
C04411=1171.245,36.733,-47.996,-179.685,6.023,148.986
C04412=1171.250,36.484,-47.981,-179.687,6.022,148.987
C04413=1171.255,36.235,-47.966,-179.690,6.021,148.988
C04414=1171.260,35.986,-47.950,-179.692,6.020,148.988
C04415=1171.265,35.736,-47.936,-179.695,6.019,148.989
C04416=1171.270,35.486,-47.920,-179.697,6.018,148.989
C04417=1171.274,35.237,-47.905,-179.700,6.017,148.990
C04418=1171.280,34.987,-47.890,-179.703,6.017,148.991
C04419=1171.285,34.737,-47.875,-179.705,6.016,148.991
C04420=1171.290,34.488,-47.860,-179.708,6.015,148.992
C04421=1171.295,34.239,-47.845,-179.711,6.014,148.992
C04422=1171.301,33.989,-47.830,-179.713,6.013,148.993
C04423=1171.305,33.740,-47.815,-179.716,6.013,148.993
C04424=1171.311,33.490,-47.799,-179.718,6.012,148.994
C04425=1171.316,33.241,-47.785,-179.721,6.011,148.995
C04426=1171.321,32.991,-47.769,-179.724,6.010,148.995
C04427=1171.326,32.742,-47.755,-179.726,6.009,148.996
C04428=1171.331,32.493,-47.740,-179.728,6.008,148.996
C04429=1171.335,32.242,-47.724,-179.731,6.008,148.997
C04430=1171.340,31.993,-47.710,-179.734,6.006,148.997
C04431=1171.346,31.743,-47.694,-179.736,6.006,148.998
C04432=1171.350,31.494,-47.679,-179.739,6.005,148.999
C04433=1171.355,31.245,-47.665,-179.741,6.004,148.999
C04434=1171.361,30.995,-47.649,-179.744,6.004,149.000
C04435=1171.366,30.745,-47.635,-179.747,6.002,149.000
C04436=1171.370,30.496,-47.620,-179.749,6.002,149.001
C04437=1171.376,30.246,-47.605,-179.752,6.001,149.002
C04438=1171.381,29.997,-47.590,-179.754,6.000,149.002
C04439=1171.386,29.748,-47.576,-179.757,6.000,149.003
C04440=1171.391,29.498,-47.560,-179.759,5.998,149.003
C04441=1171.396,29.248,-47.546,-179.762,5.998,149.004
C04442=1171.401,28.999,-47.531,-179.765,5.997,149.004
C04443=1171.406,28.749,-47.516,-179.767,5.996,149.005
C04444=1171.411,28.481,-47.501,-179.770,5.995,149.006
C04445=1171.417,28.211,-47.484,-179.773,5.995,149.006
C04446=1171.422,27.943,-47.469,-179.775,5.994,149.007
C04447=1171.427,27.674,-47.453,-179.778,5.992,149.007
C04448=1171.433,27.424,-47.437,-179.781,5.992,149.008
C04449=1171.438,27.175,-47.423,-179.783,5.991,149.009
C04450=1171.442,26.926,-47.408,-179.786,5.991,149.009
C04451=1171.447,26.676,-47.394,-179.788,5.990,149.010
C04452=1171.453,26.427,-47.378,-179.791,5.988,149.010
C04453=1171.458,26.177,-47.364,-179.794,5.988,149.011
C04454=1171.463,25.927,-47.350,-179.796,5.987,149.011
C04455=1171.468,25.678,-47.334,-179.798,5.987,149.012
C04456=1171.474,25.429,-47.320,-179.801,5.986,149.013
C04457=1171.479,25.179,-47.306,-179.803,5.985,149.013
C04458=1171.483,24.930,-47.291,-179.807,5.984,149.014
C04459=1171.488,24.680,-47.276,-179.809,5.983,149.014
C04460=1171.494,24.431,-47.261,-179.811,5.983,149.015
C04461=1171.499,24.181,-47.247,-179.814,5.982,149.016
C04462=1171.504,23.931,-47.232,-179.816,5.981,149.016
C04463=1171.508,23.682,-47.217,-179.819,5.981,149.017
C04464=1171.513,23.433,-47.203,-179.822,5.979,149.017
C04465=1171.519,23.183,-47.188,-179.824,5.979,149.018
C04466=1171.524,22.933,-47.174,-179.827,5.978,149.019
C04467=1171.528,22.684,-47.159,-179.829,5.977,149.019
C04468=1171.533,22.434,-47.145,-179.832,5.977,149.020
C04469=1171.539,22.185,-47.131,-179.834,5.976,149.020
C04470=1171.544,21.935,-47.116,-179.837,5.975,149.021
C04471=1171.549,21.686,-47.101,-179.840,5.974,149.022
C04472=1171.554,21.436,-47.087,-179.842,5.973,149.022
C04473=1171.559,21.186,-47.072,-179.844,5.973,149.023
C04474=1171.564,20.937,-47.058,-179.847,5.972,149.023
C04475=1171.569,20.688,-47.043,-179.849,5.972,149.024
C04476=1171.574,20.438,-47.029,-179.852,5.971,149.025
C04477=1171.579,20.189,-47.015,-179.855,5.969,149.025
C04478=1171.584,19.939,-47.001,-179.857,5.969,149.026
C04479=1171.590,19.689,-46.986,-179.860,5.968,149.026
C04480=1171.595,19.439,-46.971,-179.862,5.968,149.027
C04481=1171.600,19.190,-46.956,-179.865,5.967,149.028
C04482=1171.605,18.941,-46.942,-179.867,5.966,149.028
C04483=1171.609,18.691,-46.928,-179.870,5.966,149.029
C04484=1171.615,18.442,-46.914,-179.872,5.964,149.029
C04485=1171.620,18.192,-46.900,-179.875,5.964,149.030
C04486=1171.625,17.943,-46.885,-179.878,5.963,149.031
C04487=1171.630,17.693,-46.871,-179.880,5.962,149.031
C04488=1171.635,17.443,-46.857,-179.882,5.962,149.032
C04489=1171.640,17.195,-46.842,-179.885,5.961,149.032
C04490=1171.645,16.945,-46.828,-179.887,5.961,149.033
C04491=1171.650,16.695,-46.814,-179.890,5.960,149.033
C04492=1171.655,16.446,-46.799,-179.893,5.959,149.034
C04493=1171.660,16.196,-46.785,-179.895,5.958,149.035
C04494=1171.665,15.946,-46.771,-179.898,5.958,149.035
C04495=1171.670,15.697,-46.757,-179.900,5.957,149.036
C04496=1171.675,15.447,-46.743,-179.903,5.956,149.036
C04497=1171.680,15.198,-46.728,-179.905,5.955,149.037
C04498=1171.685,14.948,-46.714,-179.908,5.955,149.038
C04499=1171.691,14.699,-46.700,-179.910,5.954,149.038
C04500=1171.696,14.449,-46.686,-179.912,5.954,149.039
C04501=1171.701,14.200,-46.672,-179.916,5.952,149.039
C04502=1171.706,13.950,-46.657,-179.918,5.951,149.040
C04503=1171.711,13.701,-46.643,-179.921,5.951,149.041
C04504=1171.716,13.451,-46.629,-179.923,5.951,149.041
C04505=1171.721,13.201,-46.615,-179.925,5.950,149.042
C04506=1171.726,12.952,-46.601,-179.928,5.949,149.042
C04507=1171.732,12.703,-46.587,-179.931,5.949,149.043
C04508=1171.737,12.453,-46.572,-179.933,5.948,149.044
C04509=1171.742,12.203,-46.559,-179.935,5.947,149.044
C04510=1171.747,11.953,-46.545,-179.938,5.947,149.045
C04511=1171.752,11.704,-46.531,-179.941,5.945,149.045
C04512=1171.757,11.455,-46.517,-179.944,5.945,149.046
C04513=1171.762,11.205,-46.503,-179.946,5.944,149.046
C04514=1171.767,10.955,-46.488,-179.948,5.944,149.047
C04515=1171.772,10.706,-46.475,-179.951,5.943,149.048
C04516=1171.777,10.456,-46.460,-179.953,5.942,149.048
C04517=1171.782,10.206,-46.447,-179.956,5.942,149.049
C04518=1171.788,9.957,-46.433,-179.958,5.941,149.049
C04519=1171.793,9.707,-46.419,-179.961,5.940,149.050
C04520=1171.797,9.458,-46.405,-179.963,5.940,149.051
C04521=1171.803,9.209,-46.391,-179.965,5.939,149.051
C04522=1171.808,8.959,-46.377,-179.969,5.938,149.052
C04523=1171.813,8.709,-46.363,-179.971,5.937,149.052
C04524=1171.818,8.460,-46.349,-179.974,5.937,149.053
C04525=1171.823,8.210,-46.335,-179.976,5.936,149.054
C04526=1171.828,7.961,-46.321,-179.978,5.935,149.054
C04527=1171.833,7.711,-46.308,-179.981,5.935,149.055
C04528=1171.838,7.461,-46.294,-179.984,5.934,149.056
C04529=1171.843,7.212,-46.279,-179.986,5.933,149.056
C04530=1171.849,6.963,-46.266,-179.988,5.933,149.057
C04531=1171.853,6.713,-46.253,-179.991,5.932,149.057
C04532=1171.858,6.463,-46.238,-179.993,5.932,149.058
C04533=1171.864,6.214,-46.224,-179.996,5.931,149.059
C04534=1171.869,5.964,-46.210,-179.998,5.930,149.059
C04535=1171.873,5.714,-46.197,179.999,5.930,149.060
C04536=1171.879,5.465,-46.183,179.997,5.929,149.060
C04537=1171.884,5.216,-46.169,179.994,5.928,149.061
C04538=1171.889,4.965,-46.155,179.991,5.927,149.062
C04539=1171.894,4.717,-46.142,179.989,5.927,149.062
C04540=1171.899,4.467,-46.128,179.986,5.926,149.063
C04541=1171.905,4.217,-46.115,179.984,5.926,149.063
C04542=1171.910,3.968,-46.100,179.982,5.925,149.064
C04543=1171.914,3.718,-46.087,179.979,5.924,149.065
C04544=1171.920,3.468,-46.073,179.976,5.924,149.065
C04545=1171.925,3.219,-46.059,179.974,5.923,149.066
C04546=1171.930,2.969,-46.047,179.971,5.923,149.066
C04547=1171.935,2.720,-46.032,179.969,5.922,149.067
C04548=1171.940,2.450,-46.017,179.967,5.921,149.068
C04549=1171.946,2.182,-46.003,179.964,5.921,149.068
C04550=1171.952,1.912,-45.988,179.961,5.920,149.069
C04551=1171.957,1.642,-45.974,179.958,5.919,149.070
C04552=1171.962,1.393,-45.960,179.956,5.918,149.070
C04553=1171.968,1.143,-45.947,179.953,5.918,149.071
C04554=1171.972,0.894,-45.933,179.951,5.917,149.071
C04555=1171.977,0.645,-45.919,179.948,5.916,149.072
C04556=1171.983,0.394,-45.905,179.946,5.916,149.073
C04557=1171.987,0.146,-45.892,179.943,5.916,149.073
C04558=1171.993,-0.105,-45.879,179.941,5.915,149.074
C04559=1171.998,-0.354,-45.865,179.938,5.914,149.074
C04560=1172.003,-0.604,-45.852,179.936,5.913,149.075
C04561=1172.008,-0.853,-45.838,179.933,5.913,149.076
C04562=1172.013,-1.103,-45.825,179.931,5.912,149.076
C04563=1172.019,-1.352,-45.812,179.929,5.912,149.077
C04564=1172.024,-1.602,-45.797,179.926,5.911,149.077
C04565=1172.028,-1.852,-45.784,179.923,5.911,149.078
C04566=1172.034,-2.101,-45.770,179.921,5.910,149.079
C04567=1172.038,-2.351,-45.757,179.918,5.909,149.079
C04568=1172.044,-2.600,-45.744,179.916,5.909,149.080
C04569=1172.048,-2.850,-45.731,179.914,5.908,149.080
C04570=1172.054,-3.100,-45.717,179.911,5.908,149.081
C04571=1172.059,-3.349,-45.703,179.909,5.907,149.082
C04572=1172.064,-3.599,-45.690,179.906,5.906,149.082
C04573=1172.070,-3.848,-45.677,179.903,5.906,149.083
C04574=1172.074,-4.098,-45.664,179.901,5.905,149.083
C04575=1172.080,-4.347,-45.650,179.899,5.905,149.084
C04576=1172.084,-4.597,-45.637,179.896,5.904,149.085
C04577=1172.090,-4.846,-45.624,179.894,5.903,149.085
C04578=1172.095,-5.096,-45.611,179.891,5.903,149.086
C04579=1172.100,-5.345,-45.597,179.889,5.902,149.086
C04580=1172.105,-5.595,-45.584,179.886,5.902,149.087
C04581=1172.111,-5.845,-45.570,179.884,5.901,149.088
C04582=1172.115,-6.095,-45.557,179.882,5.900,149.088
C04583=1172.121,-6.344,-45.544,179.879,5.900,149.089
C04584=1172.125,-6.594,-45.531,179.876,5.899,149.090
C04585=1172.131,-6.844,-45.517,179.874,5.899,149.090
C04586=1172.136,-7.092,-45.504,179.871,5.898,149.091
C04587=1172.141,-7.343,-45.491,179.869,5.898,149.092
C04588=1172.146,-7.592,-45.478,179.867,5.897,149.092
C04589=1172.151,-7.842,-45.465,179.864,5.896,149.093
C04590=1172.156,-8.091,-45.451,179.862,5.896,149.093
C04591=1172.161,-8.341,-45.438,179.859,5.895,149.094
C04592=1172.167,-8.591,-45.425,179.856,5.895,149.095
C04593=1172.172,-8.840,-45.412,179.854,5.894,149.095
C04594=1172.176,-9.090,-45.399,179.852,5.893,149.096
C04595=1172.182,-9.339,-45.385,179.849,5.893,149.096
C04596=1172.187,-9.589,-45.372,179.847,5.892,149.097
C04597=1172.192,-9.839,-45.359,179.844,5.892,149.098
C04598=1172.198,-10.088,-45.347,179.841,5.891,149.098
C04599=1172.202,-10.338,-45.334,179.839,5.890,149.099
C04600=1172.208,-10.587,-45.320,179.837,5.890,149.099
C04601=1172.213,-10.836,-45.307,179.834,5.889,149.100
C04602=1172.218,-11.087,-45.294,179.832,5.889,149.101
C04603=1172.223,-11.336,-45.281,179.829,5.888,149.101
C04604=1172.228,-11.586,-45.268,179.827,5.887,149.102
C04605=1172.234,-11.836,-45.255,179.824,5.887,149.102
C04606=1172.239,-12.085,-45.242,179.822,5.886,149.103
C04607=1172.243,-12.334,-45.229,179.819,5.886,149.104
C04608=1172.249,-12.584,-45.215,179.817,5.885,149.104
C04609=1172.254,-12.833,-45.203,179.814,5.885,149.105
C04610=1172.258,-13.083,-45.190,179.812,5.884,149.105
C04611=1172.264,-13.333,-45.177,179.809,5.883,149.106
C04612=1172.269,-13.582,-45.164,179.807,5.883,149.107
C04613=1172.274,-13.832,-45.151,179.804,5.882,149.107
C04614=1172.280,-14.082,-45.138,179.802,5.882,149.108
C04615=1172.285,-14.331,-45.125,179.800,5.881,149.108
C04616=1172.289,-14.581,-45.112,179.798,5.881,149.109
C04617=1172.295,-14.831,-45.100,179.795,5.881,149.110
C04618=1172.300,-15.080,-45.087,179.793,5.880,149.110
C04619=1172.305,-15.330,-45.074,179.790,5.880,149.111
C04620=1172.310,-15.580,-45.061,179.787,5.879,149.112
C04621=1172.315,-15.829,-45.048,179.785,5.878,149.112
C04622=1172.321,-16.079,-45.035,179.783,5.878,149.113
C04623=1172.326,-16.329,-45.022,179.780,5.877,149.113
C04624=1172.331,-16.578,-45.010,179.778,5.877,149.114
C04625=1172.336,-16.827,-44.997,179.775,5.876,149.115
C04626=1172.341,-17.078,-44.983,179.773,5.875,149.115
C04627=1172.346,-17.327,-44.971,179.770,5.875,149.116
C04628=1172.351,-17.576,-44.958,179.768,5.874,149.117
C04629=1172.356,-17.826,-44.946,179.765,5.874,149.117
C04630=1172.362,-18.076,-44.932,179.763,5.873,149.118
C04631=1172.367,-18.326,-44.920,179.760,5.873,149.118
C04632=1172.372,-18.575,-44.908,179.758,5.872,149.119
C04633=1172.377,-18.824,-44.895,179.756,5.872,149.120
C04634=1172.382,-19.074,-44.882,179.754,5.871,149.120
C04635=1172.388,-19.324,-44.869,179.751,5.871,149.121
C04636=1172.393,-19.573,-44.856,179.748,5.870,149.121
C04637=1172.398,-19.823,-44.844,179.746,5.870,149.122
C04638=1172.403,-20.073,-44.831,179.744,5.869,149.123
C04639=1172.408,-20.323,-44.819,179.741,5.869,149.123
C04640=1172.413,-20.572,-44.806,179.739,5.868,149.124
C04641=1172.419,-20.822,-44.793,179.736,5.867,149.124
C04642=1172.424,-21.071,-44.780,179.733,5.867,149.125
C04643=1172.429,-21.321,-44.767,179.731,5.866,149.126
C04644=1172.434,-21.571,-44.756,179.729,5.866,149.126
C04645=1172.439,-21.820,-44.743,179.727,5.866,149.127
C04646=1172.444,-22.070,-44.730,179.724,5.865,149.127
C04647=1172.449,-22.320,-44.717,179.722,5.865,149.128
C04648=1172.454,-22.569,-44.705,179.719,5.864,149.129
C04649=1172.460,-22.819,-44.692,179.717,5.864,149.129
C04650=1172.465,-23.068,-44.680,179.714,5.863,149.130
C04651=1172.470,-23.318,-44.667,179.712,5.862,149.130
C04652=1172.475,-23.587,-44.653,179.709,5.862,149.131
C04653=1172.481,-23.858,-44.640,179.707,5.861,149.132
C04654=1172.487,-24.127,-44.626,179.704,5.861,149.133
C04655=1172.492,-24.397,-44.613,179.701,5.861,149.133
C04656=1172.497,-24.647,-44.601,179.699,5.860,149.134
C04657=1172.503,-24.896,-44.588,179.696,5.859,149.134
C04658=1172.508,-25.145,-44.576,179.694,5.859,149.135
C04659=1172.512,-25.396,-44.563,179.692,5.858,149.136
C04660=1172.518,-25.645,-44.551,179.689,5.858,149.136
C04661=1172.523,-25.895,-44.538,179.687,5.857,149.137
C04662=1172.528,-26.145,-44.526,179.685,5.857,149.137
C04663=1172.533,-26.394,-44.514,179.682,5.857,149.138
C04664=1172.538,-26.643,-44.501,179.680,5.856,149.139
C04665=1172.544,-26.893,-44.489,179.677,5.855,149.139
C04666=1172.548,-27.143,-44.476,179.675,5.855,149.140
C04667=1172.554,-27.393,-44.464,179.672,5.854,149.140
C04668=1172.559,-27.643,-44.452,179.670,5.854,149.141
C04669=1172.564,-27.892,-44.439,179.667,5.853,149.142
C04670=1172.569,-28.142,-44.427,179.665,5.852,149.142
C04671=1172.575,-28.391,-44.415,179.663,5.853,149.143
C04672=1172.580,-28.641,-44.403,179.661,5.852,149.144
C04673=1172.585,-28.890,-44.390,179.658,5.852,149.144
C04674=1172.590,-29.140,-44.378,179.655,5.851,149.145
C04675=1172.595,-29.390,-44.365,179.653,5.850,149.145
C04676=1172.600,-29.640,-44.353,179.650,5.850,149.146
C04677=1172.606,-29.890,-44.341,179.648,5.849,149.147
C04678=1172.611,-30.139,-44.328,179.646,5.849,149.147
C04679=1172.616,-30.389,-44.316,179.644,5.849,149.148
C04680=1172.621,-30.638,-44.304,179.641,5.848,149.148
C04681=1172.627,-30.888,-44.292,179.639,5.848,149.149
C04682=1172.632,-31.137,-44.279,179.636,5.847,149.150
C04683=1172.637,-31.387,-44.267,179.634,5.847,149.150
C04684=1172.642,-31.637,-44.255,179.631,5.846,149.151
C04685=1172.647,-31.886,-44.244,179.629,5.846,149.152
C04686=1172.652,-32.136,-44.231,179.627,5.846,149.152
C04687=1172.658,-32.386,-44.219,179.624,5.845,149.153
C04688=1172.663,-32.635,-44.207,179.622,5.845,149.154
C04689=1172.668,-32.885,-44.195,179.619,5.844,149.154
C04690=1172.673,-33.134,-44.182,179.617,5.844,149.155
C04691=1172.678,-33.385,-44.170,179.615,5.843,149.155
C04692=1172.684,-33.635,-44.158,179.612,5.842,149.156
C04693=1172.688,-33.884,-44.146,179.610,5.843,149.157
C04694=1172.693,-34.134,-44.134,179.608,5.842,149.157
C04695=1172.699,-34.383,-44.121,179.605,5.841,149.158
C04696=1172.704,-34.633,-44.110,179.602,5.841,149.158
C04697=1172.709,-34.883,-44.098,179.600,5.840,149.159
C04698=1172.715,-35.132,-44.085,179.598,5.840,149.160
C04699=1172.720,-35.382,-44.073,179.595,5.839,149.160
C04700=1172.724,-35.631,-44.061,179.593,5.839,149.161
C04701=1172.730,-35.881,-44.049,179.591,5.839,149.161
C04702=1172.735,-36.131,-44.037,179.588,5.838,149.162
C04703=1172.740,-36.380,-44.025,179.586,5.838,149.163
C04704=1172.746,-36.630,-44.013,179.583,5.837,149.163
C04705=1172.750,-36.880,-44.002,179.581,5.836,149.164
C04706=1172.756,-37.129,-43.989,179.579,5.837,149.165
C04707=1172.761,-37.379,-43.977,179.577,5.836,149.165
C04708=1172.767,-37.628,-43.966,179.574,5.835,149.166
C04709=1172.772,-37.878,-43.954,179.571,5.835,149.166
C04710=1172.777,-38.127,-43.942,179.569,5.834,149.167
C04711=1172.782,-38.377,-43.930,179.566,5.834,149.168
C04712=1172.788,-38.627,-43.918,179.564,5.834,149.168
C04713=1172.793,-38.876,-43.905,179.562,5.833,149.169
C04714=1172.798,-39.126,-43.894,179.560,5.833,149.169
C04715=1172.803,-39.376,-43.882,179.557,5.832,149.170
C04716=1172.808,-39.626,-43.870,179.555,5.832,149.171
C04717=1172.813,-39.875,-43.858,179.552,5.831,149.171
C04718=1172.818,-40.125,-43.846,179.550,5.831,149.172
C04719=1172.824,-40.375,-43.834,179.548,5.831,149.172
C04720=1172.829,-40.625,-43.823,179.545,5.830,149.173
C04721=1172.834,-40.874,-43.811,179.543,5.830,149.174
C04722=1172.839,-41.124,-43.799,179.540,5.829,149.174
C04723=1172.844,-41.374,-43.787,179.538,5.828,149.175
C04724=1172.850,-41.623,-43.776,179.536,5.829,149.176
C04725=1172.855,-41.872,-43.764,179.533,5.828,149.176
C04726=1172.860,-42.122,-43.752,179.531,5.827,149.177
C04727=1172.865,-42.372,-43.741,179.529,5.827,149.177
C04728=1172.870,-42.621,-43.728,179.526,5.827,149.178
C04729=1172.876,-42.871,-43.716,179.524,5.827,149.179
C04730=1172.880,-43.121,-43.705,179.522,5.826,149.179
C04731=1172.886,-43.371,-43.693,179.519,5.825,149.180
C04732=1172.891,-43.621,-43.681,179.517,5.825,149.180
C04733=1172.896,-43.870,-43.670,179.514,5.825,149.181
C04734=1172.902,-44.120,-43.658,179.513,5.824,149.182
C04735=1172.907,-44.370,-43.647,179.510,5.824,149.182
C04736=1172.912,-44.619,-43.635,179.507,5.824,149.183
C04737=1172.917,-44.869,-43.623,179.505,5.823,149.184
C04738=1172.922,-45.118,-43.611,179.502,5.822,149.184
C04739=1172.927,-45.368,-43.600,179.501,5.822,149.185
C04740=1172.933,-45.618,-43.588,179.498,5.822,149.185
C04741=1172.938,-45.867,-43.577,179.495,5.822,149.186
C04742=1172.944,-46.117,-43.565,179.493,5.821,149.187
C04743=1172.948,-46.367,-43.554,179.491,5.820,149.187
C04744=1172.954,-46.616,-43.542,179.489,5.820,149.188
C04745=1172.959,-46.866,-43.530,179.486,5.820,149.188
C04746=1172.964,-47.116,-43.518,179.484,5.819,149.189
C04747=1172.970,-47.365,-43.507,179.481,5.819,149.190
C04748=1172.974,-47.615,-43.496,179.479,5.818,149.190
C04749=1172.980,-47.865,-43.484,179.477,5.819,149.191
C04750=1172.985,-48.114,-43.473,179.475,5.818,149.192
C04751=1172.990,-48.364,-43.461,179.472,5.817,149.192
C04752=1172.995,-48.614,-43.449,179.470,5.817,149.193
C04753=1173.001,-48.863,-43.438,179.467,5.816,149.193
C04754=1173.006,-49.113,-43.426,179.465,5.817,149.194
C04755=1173.011,-49.363,-43.415,179.463,5.816,149.195
C04756=1173.016,-49.634,-43.402,179.460,5.815,149.195
C04757=1173.022,-49.903,-43.390,179.457,5.815,149.196
C04758=1173.028,-50.174,-43.378,179.455,5.814,149.197
C04759=1173.034,-50.444,-43.365,179.453,5.814,149.197
C04760=1173.039,-50.694,-43.354,179.450,5.813,149.198
C04761=1173.044,-50.944,-43.342,179.448,5.814,149.199
C04762=1173.049,-51.194,-43.331,179.446,5.813,149.199
C04763=1173.054,-51.444,-43.319,179.443,5.812,149.200
C04764=1173.060,-51.693,-43.308,179.440,5.812,149.200
C04765=1173.065,-51.943,-43.296,179.439,5.812,149.201
C04766=1173.070,-52.192,-43.285,179.436,5.812,149.202
C04767=1173.075,-52.442,-43.273,179.434,5.811,149.202
C04768=1173.081,-52.691,-43.262,179.431,5.810,149.203
C04769=1173.086,-52.941,-43.252,179.429,5.811,149.204
C04770=1173.091,-53.191,-43.240,179.427,5.810,149.204
C04771=1173.096,-53.441,-43.229,179.424,5.809,149.205
C04772=1173.102,-53.690,-43.217,179.422,5.809,149.205
C04773=1173.106,-53.940,-43.206,179.419,5.808,149.206
C04774=1173.112,-54.190,-43.195,179.417,5.809,149.207
C04775=1173.117,-54.440,-43.183,179.415,5.808,149.207
C04776=1173.122,-54.689,-43.172,179.412,5.807,149.208
C04777=1173.128,-54.939,-43.161,179.410,5.807,149.208
C04778=1173.132,-55.188,-43.149,179.408,5.807,149.209
C04779=1173.137,-55.439,-43.139,179.406,5.807,149.210
C04780=1173.143,-55.688,-43.127,179.403,5.806,149.210
C04781=1173.148,-55.938,-43.116,179.401,5.805,149.211
C04782=1173.153,-56.188,-43.104,179.399,5.805,149.211
C04783=1173.159,-56.437,-43.094,179.396,5.805,149.212
C04784=1173.164,-56.687,-43.083,179.394,5.805,149.213
C04785=1173.169,-56.937,-43.071,179.392,5.804,149.213
C04786=1173.174,-57.186,-43.060,179.390,5.804,149.214
C04787=1173.179,-57.436,-43.049,179.387,5.803,149.214
C04788=1173.185,-57.686,-43.037,179.385,5.803,149.215
C04789=1173.190,-57.935,-43.026,179.382,5.802,149.216
C04790=1173.195,-58.185,-43.016,179.380,5.802,149.216
C04791=1173.201,-58.435,-43.004,179.378,5.802,149.217
C04792=1173.205,-58.684,-42.993,179.376,5.801,149.217
C04793=1173.211,-58.934,-42.982,179.373,5.802,149.218
C04794=1173.216,-59.184,-42.970,179.371,5.801,149.219
C04795=1173.221,-59.434,-42.959,179.369,5.800,149.219
C04796=1173.227,-59.683,-42.949,179.366,5.800,149.220
C04797=1173.231,-59.933,-42.938,179.364,5.800,149.221
C04798=1173.237,-60.183,-42.926,179.362,5.800,149.221
C04799=1173.242,-60.432,-42.916,179.359,5.799,149.222
C04800=1173.247,-60.682,-42.904,179.357,5.798,149.222
C04801=1173.253,-60.932,-42.893,179.355,5.799,149.223
C04802=1173.258,-61.181,-42.882,179.353,5.798,149.224
C04803=1173.263,-61.431,-42.871,179.350,5.798,149.224
C04804=1173.268,-61.681,-42.861,179.348,5.798,149.225
C04805=1173.274,-61.930,-42.849,179.346,5.797,149.225
C04806=1173.279,-62.181,-42.838,179.343,5.797,149.226
C04807=1173.284,-62.430,-42.827,179.341,5.796,149.227
C04808=1173.289,-62.680,-42.817,179.339,5.796,149.227
C04809=1173.295,-62.929,-42.805,179.337,5.795,149.228
C04810=1173.300,-63.179,-42.794,179.334,5.795,149.229
C04811=1173.305,-63.429,-42.783,179.331,5.795,149.229
C04812=1173.310,-63.678,-42.772,179.330,5.795,149.230
C04813=1173.315,-63.928,-42.762,179.327,5.794,149.230
C04814=1173.321,-64.177,-42.750,179.325,5.793,149.231
C04815=1173.326,-64.428,-42.740,179.323,5.794,149.232
C04816=1173.331,-64.677,-42.728,179.320,5.793,149.232
C04817=1173.336,-64.927,-42.718,179.318,5.793,149.233
C04818=1173.341,-65.176,-42.707,179.315,5.792,149.234
C04819=1173.347,-65.426,-42.696,179.314,5.792,149.234
C04820=1173.352,-65.676,-42.685,179.311,5.792,149.235
C04821=1173.357,-65.926,-42.674,179.309,5.791,149.235
C04822=1173.363,-66.176,-42.664,179.307,5.791,149.236
C04823=1173.367,-66.425,-42.653,179.304,5.791,149.237
C04824=1173.373,-66.675,-42.643,179.302,5.790,149.237
C04825=1173.378,-66.925,-42.631,179.300,5.791,149.238
C04826=1173.384,-67.174,-42.621,179.297,5.790,149.238
C04827=1173.389,-67.424,-42.609,179.295,5.789,149.239
C04828=1173.394,-67.673,-42.599,179.293,5.789,149.239
C04829=1173.399,-67.924,-42.588,179.291,5.789,149.240
C04830=1173.405,-68.173,-42.578,179.288,5.789,149.241
C04831=1173.410,-68.423,-42.567,179.286,5.788,149.241
C04832=1173.415,-68.672,-42.556,179.284,5.788,149.242
C04833=1173.421,-68.922,-42.545,179.281,5.787,149.243
C04834=1173.426,-69.173,-42.534,179.279,5.787,149.243
C04835=1173.431,-69.422,-42.523,179.277,5.787,149.244
C04836=1173.436,-69.672,-42.513,179.274,5.787,149.244
C04837=1173.442,-69.921,-42.503,179.272,5.786,149.245
C04838=1173.446,-70.171,-42.491,179.270,5.786,149.246
C04839=1173.452,-70.421,-42.481,179.268,5.786,149.246
C04840=1173.457,-70.671,-42.470,179.265,5.785,149.247
C04841=1173.462,-70.920,-42.460,179.263,5.785,149.248
C04842=1173.467,-71.170,-42.449,179.261,5.785,149.248
C04843=1173.473,-71.419,-42.439,179.258,5.784,149.249
C04844=1173.478,-71.669,-42.427,179.256,5.784,149.249
C04845=1173.484,-71.919,-42.417,179.254,5.784,149.250
C04846=1173.489,-72.168,-42.406,179.251,5.783,149.251
C04847=1173.494,-72.419,-42.396,179.249,5.783,149.251
C04848=1173.500,-72.668,-42.385,179.247,5.783,149.252
C04849=1173.505,-72.918,-42.374,179.245,5.782,149.252
C04850=1173.510,-73.167,-42.364,179.242,5.782,149.253
C04851=1173.515,-73.418,-42.354,179.241,5.782,149.253
C04852=1173.520,-73.667,-42.343,179.238,5.781,149.254
C04853=1173.525,-73.917,-42.332,179.235,5.781,149.255
C04854=1173.531,-74.166,-42.322,179.234,5.781,149.255
C04855=1173.536,-74.417,-42.311,179.231,5.781,149.256
C04856=1173.541,-74.666,-42.300,179.229,5.780,149.257
C04857=1173.547,-74.915,-42.290,179.227,5.780,149.257
C04858=1173.552,-75.165,-42.280,179.225,5.779,149.258
C04859=1173.558,-75.415,-42.269,179.222,5.779,149.258
C04860=1173.563,-75.686,-42.258,179.219,5.779,149.259
C04861=1173.568,-75.957,-42.246,179.218,5.779,149.260
C04862=1173.575,-76.228,-42.235,179.215,5.778,149.260
C04863=1173.580,-76.499,-42.224,179.212,5.778,149.261
C04864=1173.586,-76.749,-42.214,179.210,5.777,149.262
C04865=1173.590,-76.999,-42.203,179.208,5.777,149.262
C04866=1173.596,-77.248,-42.192,179.205,5.777,149.263
C04867=1173.601,-77.498,-42.182,179.203,5.776,149.263
C04868=1173.607,-77.748,-42.172,179.201,5.777,149.264
C04869=1173.612,-77.997,-42.161,179.199,5.776,149.265
C04870=1173.617,-78.248,-42.151,179.196,5.775,149.265
C04871=1173.623,-78.497,-42.141,179.195,5.775,149.266
C04872=1173.628,-78.747,-42.130,179.192,5.775,149.267
C04873=1173.633,-78.997,-42.120,179.191,5.775,149.267
C04874=1173.638,-79.246,-42.110,179.188,5.775,149.268
C04875=1173.643,-79.496,-42.099,179.185,5.774,149.268
C04876=1173.648,-79.745,-42.089,179.184,5.774,149.269
C04877=1173.654,-79.995,-42.079,179.181,5.774,149.270
C04878=1173.659,-80.245,-42.068,179.179,5.773,149.270
C04879=1173.665,-80.495,-42.058,179.177,5.773,149.271
C04880=1173.670,-80.745,-42.047,179.174,5.773,149.271
C04881=1173.675,-80.995,-42.037,179.172,5.772,149.272
C04882=1173.680,-81.244,-42.027,179.170,5.772,149.272
C04883=1173.685,-81.494,-42.017,179.167,5.772,149.273
C04884=1173.691,-81.744,-42.007,179.165,5.771,149.274
C04885=1173.696,-81.993,-41.996,179.163,5.771,149.274
C04886=1173.701,-82.243,-41.986,179.161,5.771,149.275
C04887=1173.707,-82.493,-41.976,179.158,5.770,149.276
C04888=1173.712,-82.742,-41.966,179.157,5.770,149.276
C04889=1173.717,-82.992,-41.955,179.154,5.770,149.277
C04890=1173.722,-83.242,-41.945,179.152,5.770,149.277
C04891=1173.728,-83.491,-41.935,179.150,5.769,149.278
C04892=1173.733,-83.742,-41.924,179.147,5.769,149.279
C04893=1173.739,-83.991,-41.914,179.146,5.769,149.279
C04894=1173.743,-84.240,-41.905,179.143,5.769,149.280
C04895=1173.748,-84.491,-41.894,179.141,5.768,149.280
C04896=1173.754,-84.740,-41.884,179.139,5.768,149.281
C04897=1173.760,-84.990,-41.874,179.136,5.768,149.282
C04898=1173.764,-85.240,-41.864,179.134,5.768,149.282
C04899=1173.770,-85.490,-41.854,179.132,5.767,149.283
C04900=1173.775,-85.739,-41.844,179.129,5.767,149.283
C04901=1173.781,-85.989,-41.834,179.128,5.767,149.284
C04902=1173.785,-86.239,-41.824,179.125,5.766,149.285
C04903=1173.791,-86.488,-41.814,179.123,5.766,149.285
C04904=1173.796,-86.738,-41.803,179.121,5.766,149.286
C04905=1173.801,-86.988,-41.793,179.119,5.765,149.286
C04906=1173.806,-87.237,-41.783,179.117,5.766,149.287
C04907=1173.812,-87.488,-41.774,179.114,5.765,149.287
C04908=1173.818,-87.737,-41.763,179.112,5.764,149.288
C04909=1173.823,-87.987,-41.753,179.110,5.764,149.289
C04910=1173.828,-88.237,-41.743,179.108,5.764,149.289
C04911=1173.833,-88.486,-41.733,179.105,5.764,149.290
C04912=1173.839,-88.736,-41.723,179.103,5.764,149.291
C04913=1173.843,-88.986,-41.714,179.101,5.763,149.291
C04914=1173.849,-89.236,-41.703,179.099,5.763,149.292
C04915=1173.855,-89.485,-41.693,179.096,5.763,149.292
C04916=1173.860,-89.735,-41.683,179.094,5.762,149.293
C04917=1173.864,-89.985,-41.673,179.092,5.762,149.294
C04918=1173.870,-90.235,-41.663,179.090,5.762,149.294
C04919=1173.876,-90.485,-41.653,179.088,5.762,149.295
C04920=1173.881,-90.734,-41.644,179.086,5.761,149.295
C04921=1173.886,-90.984,-41.633,179.083,5.761,149.296
C04922=1173.892,-91.234,-41.624,179.081,5.761,149.297
C04923=1173.897,-91.483,-41.614,179.079,5.761,149.297
C04924=1173.902,-91.733,-41.604,179.077,5.761,149.298
C04925=1173.907,-91.982,-41.594,179.074,5.760,149.298
C04926=1173.912,-92.233,-41.584,179.072,5.759,149.299
C04927=1173.918,-92.483,-41.574,179.070,5.760,149.300
C04928=1173.923,-92.732,-41.564,179.068,5.759,149.300
C04929=1173.929,-92.982,-41.555,179.066,5.759,149.301
C04930=1173.934,-93.232,-41.544,179.064,5.759,149.301
C04931=1173.939,-93.481,-41.535,179.061,5.758,149.302
C04932=1173.944,-93.731,-41.525,179.059,5.758,149.303
C04933=1173.950,-93.981,-41.515,179.057,5.758,149.303
C04934=1173.955,-94.230,-41.505,179.055,5.758,149.304
C04935=1173.961,-94.480,-41.495,179.052,5.758,149.304
C04936=1173.965,-94.731,-41.486,179.050,5.757,149.305
C04937=1173.971,-94.980,-41.476,179.048,5.757,149.306
C04938=1173.976,-95.230,-41.467,179.046,5.756,149.306
C04939=1173.981,-95.479,-41.457,179.044,5.756,149.307
C04940=1173.987,-95.729,-41.446,179.042,5.756,149.307
C04941=1173.992,-95.979,-41.438,179.040,5.755,149.308
C04942=1173.997,-96.229,-41.427,179.037,5.756,149.308
C04943=1174.002,-96.478,-41.417,179.035,5.755,149.309
C04944=1174.008,-96.728,-41.408,179.033,5.755,149.310
C04945=1174.013,-96.978,-41.398,179.031,5.754,149.310
C04946=1174.019,-97.228,-41.389,179.029,5.755,149.311
C04947=1174.024,-97.477,-41.379,179.027,5.754,149.311
C04948=1174.029,-97.727,-41.369,179.024,5.754,149.312
C04949=1174.035,-97.978,-41.359,179.022,5.754,149.313
C04950=1174.039,-98.227,-41.349,179.020,5.753,149.313
C04951=1174.045,-98.477,-41.340,179.018,5.753,149.314
C04952=1174.050,-98.726,-41.330,179.015,5.753,149.314
C04953=1174.056,-98.976,-41.321,179.014,5.753,149.315
C04954=1174.061,-99.226,-41.311,179.011,5.753,149.316
C04955=1174.067,-99.476,-41.302,179.009,5.752,149.316
C04956=1174.072,-99.725,-41.292,179.007,5.752,149.317
C04957=1174.078,-99.975,-41.283,179.005,5.751,149.317
C04958=1174.082,-100.225,-41.273,179.003,5.752,149.318
C04959=1174.088,-100.475,-41.263,179.000,5.751,149.319
C04960=1174.093,-100.724,-41.254,178.998,5.751,149.319
C04961=1174.099,-100.975,-41.244,178.996,5.751,149.320
C04962=1174.103,-101.224,-41.234,178.994,5.750,149.320
C04963=1174.109,-101.474,-41.225,178.992,5.750,149.321
C04964=1174.115,-101.746,-41.215,178.989,5.750,149.322
C04965=1174.120,-102.017,-41.204,178.987,5.749,149.322
C04966=1174.126,-102.288,-41.194,178.985,5.750,149.323
C04967=1174.132,-102.560,-41.184,178.982,5.749,149.324
C04968=1174.137,-102.811,-41.174,178.980,5.748,149.324
C04969=1174.142,-103.060,-41.165,178.978,5.749,149.325
C04970=1174.148,-103.310,-41.155,178.976,5.748,149.325
C04971=1174.153,-103.559,-41.145,178.974,5.748,149.326
C04972=1174.158,-103.810,-41.136,178.972,5.748,149.326
C04973=1174.164,-104.060,-41.127,178.970,5.748,149.327
C04974=1174.168,-104.309,-41.117,178.967,5.747,149.328
C04975=1174.174,-104.559,-41.108,178.966,5.747,149.328
C04976=1174.179,-104.808,-41.098,178.963,5.747,149.329
C04977=1174.185,-105.059,-41.089,178.961,5.746,149.329
C04978=1174.190,-105.309,-41.080,178.959,5.747,149.330
C04979=1174.195,-105.558,-41.070,178.957,5.746,149.331
C04980=1174.201,-105.808,-41.061,178.955,5.746,149.331
C04981=1174.206,-106.058,-41.052,178.952,5.745,149.332
C04982=1174.211,-106.307,-41.042,178.951,5.745,149.332
C04983=1174.217,-106.557,-41.033,178.948,5.745,149.333
C04984=1174.222,-106.807,-41.024,178.946,5.745,149.333
C04985=1174.227,-107.056,-41.014,178.944,5.745,149.334
C04986=1174.233,-107.306,-41.005,178.942,5.745,149.335
C04987=1174.238,-107.556,-40.996,178.939,5.744,149.335
C04988=1174.244,-107.806,-40.985,178.937,5.744,149.336
C04989=1174.249,-108.056,-40.977,178.936,5.744,149.336
C04990=1174.254,-108.305,-40.968,178.933,5.743,149.337
C04991=1174.260,-108.555,-40.957,178.931,5.743,149.337
C04992=1174.265,-108.805,-40.949,178.929,5.743,149.338
C04993=1174.270,-109.055,-40.940,178.927,5.743,149.339
C04994=1174.275,-109.305,-40.931,178.924,5.743,149.339
C04995=1174.281,-109.554,-40.920,178.923,5.743,149.340
C04996=1174.286,-109.804,-40.912,178.921,5.742,149.340
C04997=1174.291,-110.054,-40.903,178.919,5.742,149.341
C04998=1174.297,-110.304,-40.893,178.916,5.741,149.342
C04999=1174.302,-110.553,-40.884,178.914,5.741,149.342
C05000=1174.307,-110.803,-40.875,178.912,5.741,149.343
C05001=1174.313,-111.053,-40.865,178.909,5.741,149.343
C05002=1174.318,-111.303,-40.856,178.908,5.741,149.344
C05003=1174.323,-111.552,-40.847,178.906,5.740,149.344
C05004=1174.328,-111.802,-40.838,178.904,5.740,149.345
C05005=1174.334,-112.052,-40.828,178.901,5.740,149.346
C05006=1174.339,-112.302,-40.819,178.899,5.740,149.346
C05007=1174.345,-112.551,-40.811,178.897,5.739,149.347
C05008=1174.350,-112.801,-40.802,178.895,5.740,149.348
C05009=1174.356,-113.051,-40.792,178.893,5.739,149.348
C05010=1174.361,-113.301,-40.783,178.891,5.739,149.349
C05011=1174.366,-113.550,-40.774,178.889,5.738,149.349
C05012=1174.371,-113.800,-40.765,178.887,5.739,149.350
C05013=1174.377,-114.050,-40.756,178.884,5.738,149.350
C05014=1174.382,-114.300,-40.747,178.883,5.738,149.351
C05015=1174.387,-114.550,-40.737,178.880,5.737,149.351
C05016=1174.392,-114.799,-40.728,178.878,5.738,149.352
C05017=1174.397,-115.049,-40.719,178.876,5.737,149.353
C05018=1174.403,-115.299,-40.710,178.873,5.737,149.353
C05019=1174.408,-115.549,-40.701,178.872,5.737,149.354
C05020=1174.414,-115.798,-40.692,178.870,5.736,149.354
C05021=1174.419,-116.048,-40.683,178.868,5.736,149.355
C05022=1174.425,-116.298,-40.675,178.865,5.736,149.356
C05023=1174.430,-116.548,-40.665,178.863,5.736,149.356
C05024=1174.436,-116.798,-40.656,178.861,5.735,149.357
C05025=1174.441,-117.047,-40.647,178.860,5.735,149.357
C05026=1174.446,-117.297,-40.638,178.857,5.735,149.358
C05027=1174.451,-117.547,-40.629,178.855,5.735,149.358
C05028=1174.456,-117.797,-40.620,178.853,5.735,149.359
C05029=1174.463,-118.046,-40.611,178.851,5.735,149.360
C05030=1174.468,-118.296,-40.602,178.849,5.734,149.360
C05031=1174.473,-118.546,-40.593,178.847,5.734,149.361
C05032=1174.478,-118.796,-40.584,178.845,5.733,149.361
C05033=1174.483,-119.046,-40.575,178.843,5.733,149.362
C05034=1174.488,-119.296,-40.566,178.840,5.733,149.363
C05035=1174.494,-119.545,-40.557,178.839,5.733,149.363
C05036=1174.499,-119.795,-40.549,178.836,5.733,149.364
C05037=1174.505,-120.045,-40.539,178.834,5.733,149.364
C05038=1174.510,-120.295,-40.530,178.832,5.732,149.365
C05039=1174.516,-120.544,-40.522,178.830,5.732,149.365
C05040=1174.521,-120.794,-40.513,178.828,5.732,149.366
C05041=1174.526,-121.044,-40.504,178.826,5.732,149.366
C05042=1174.532,-121.293,-40.495,178.824,5.731,149.367
C05043=1174.537,-121.543,-40.486,178.822,5.731,149.368
C05044=1174.542,-121.793,-40.477,178.819,5.731,149.368
C05045=1174.547,-122.043,-40.468,178.818,5.731,149.369
C05046=1174.552,-122.293,-40.460,178.816,5.730,149.369
C05047=1174.558,-122.543,-40.451,178.813,5.731,149.370
C05048=1174.564,-122.792,-40.443,178.811,5.730,149.370
C05049=1174.569,-123.042,-40.434,178.810,5.730,149.371
C05050=1174.575,-123.292,-40.424,178.807,5.730,149.372
C05051=1174.580,-123.542,-40.416,178.805,5.730,149.372
C05052=1174.585,-123.792,-40.407,178.803,5.729,149.373
C05053=1174.591,-124.041,-40.398,178.801,5.729,149.373
C05054=1174.596,-124.291,-40.389,178.799,5.728,149.374
C05055=1174.601,-124.541,-40.380,178.797,5.729,149.375
C05056=1174.606,-124.791,-40.371,178.795,5.728,149.375
C05057=1174.612,-125.041,-40.363,178.793,5.728,149.376
C05058=1174.617,-125.290,-40.355,178.790,5.728,149.376
C05059=1174.623,-125.540,-40.346,178.789,5.728,149.377
C05060=1174.628,-125.790,-40.337,178.787,5.727,149.377
C05061=1174.633,-126.040,-40.328,178.784,5.727,149.378
C05062=1174.639,-126.289,-40.320,178.782,5.727,149.378
C05063=1174.644,-126.540,-40.311,178.781,5.727,149.379
C05064=1174.649,-126.789,-40.302,178.779,5.727,149.380
C05065=1174.655,-127.039,-40.294,178.776,5.726,149.380
C05066=1174.660,-127.289,-40.285,178.775,5.726,149.381
C05067=1174.665,-127.538,-40.276,178.772,5.726,149.381
C05068=1174.244,-127.550,-40.317,178.768,5.729,149.383
C05069=1174.239,-127.300,-40.325,178.771,5.730,149.382
C05070=1174.233,-127.050,-40.334,178.773,5.730,149.382
C05071=1174.228,-126.800,-40.343,178.775,5.730,149.381
C05072=1174.222,-126.551,-40.351,178.777,5.730,149.381
C05073=1174.217,-126.301,-40.360,178.779,5.731,149.380
C05074=1174.212,-126.051,-40.369,178.781,5.731,149.380
C05075=1174.207,-125.801,-40.377,178.783,5.731,149.379
C05076=1174.201,-125.552,-40.386,178.785,5.731,149.379
C05077=1174.196,-125.302,-40.395,178.787,5.732,149.378
C05078=1174.191,-125.052,-40.404,178.789,5.731,149.377
C05079=1174.185,-124.802,-40.413,178.791,5.732,149.377
C05080=1174.180,-124.552,-40.422,178.793,5.732,149.376
C05081=1174.174,-124.303,-40.430,178.796,5.732,149.376
C05082=1174.169,-124.052,-40.438,178.797,5.732,149.375
C05083=1174.164,-123.803,-40.447,178.799,5.733,149.375
C05084=1174.159,-123.553,-40.456,178.801,5.733,149.374
C05085=1174.153,-123.303,-40.465,178.804,5.734,149.374
C05086=1174.147,-123.053,-40.474,178.805,5.734,149.373
C05087=1174.142,-122.804,-40.483,178.808,5.734,149.372
C05088=1174.137,-122.554,-40.492,178.810,5.734,149.372
C05089=1174.131,-122.304,-40.501,178.812,5.734,149.371
C05090=1174.126,-122.054,-40.510,178.814,5.734,149.371
C05091=1174.121,-121.805,-40.518,178.816,5.735,149.370
C05092=1174.115,-121.555,-40.527,178.818,5.735,149.369
C05093=1174.110,-121.305,-40.536,178.820,5.735,149.369
C05094=1174.105,-121.055,-40.544,178.822,5.735,149.368
C05095=1174.100,-120.805,-40.553,178.825,5.736,149.368
C05096=1174.094,-120.555,-40.562,178.826,5.736,149.367
C05097=1174.089,-120.306,-40.570,178.829,5.736,149.367
C05098=1174.083,-120.056,-40.579,178.830,5.736,149.366
C05099=1174.078,-119.806,-40.589,178.833,5.737,149.366
C05100=1174.072,-119.556,-40.598,178.835,5.736,149.365
C05101=1174.067,-119.306,-40.607,178.837,5.737,149.364
C05102=1174.062,-119.056,-40.616,178.839,5.737,149.364
C05103=1174.057,-118.806,-40.624,178.841,5.737,149.363
C05104=1174.051,-118.557,-40.633,178.843,5.737,149.363
C05105=1174.046,-118.307,-40.642,178.846,5.738,149.362
C05106=1174.041,-118.058,-40.651,178.847,5.738,149.361
C05107=1174.035,-117.807,-40.660,178.849,5.739,149.361
C05108=1174.030,-117.558,-40.670,178.851,5.738,149.360
C05109=1174.025,-117.308,-40.679,178.854,5.739,149.360
C05110=1174.020,-117.059,-40.688,178.855,5.739,149.359
C05111=1174.015,-116.809,-40.697,178.858,5.739,149.359
C05112=1174.009,-116.560,-40.705,178.859,5.739,149.358
C05113=1174.004,-116.310,-40.714,178.862,5.740,149.357
C05114=1173.998,-116.060,-40.724,178.864,5.740,149.357
C05115=1173.993,-115.810,-40.732,178.866,5.740,149.356
C05116=1173.987,-115.560,-40.741,178.868,5.740,149.356
C05117=1173.982,-115.310,-40.750,178.870,5.741,149.355
C05118=1173.977,-115.060,-40.759,178.872,5.740,149.354
C05119=1173.971,-114.810,-40.769,178.874,5.741,149.354
C05120=1173.966,-114.561,-40.778,178.876,5.741,149.354
C05121=1173.961,-114.311,-40.787,178.879,5.741,149.353
C05122=1173.955,-114.062,-40.796,178.880,5.741,149.352
C05123=1173.949,-113.812,-40.805,178.883,5.742,149.352
C05124=1173.944,-113.562,-40.814,178.885,5.742,149.351
C05125=1173.939,-113.312,-40.823,178.887,5.742,149.351
C05126=1173.934,-113.062,-40.832,178.889,5.742,149.350
C05127=1173.929,-112.813,-40.841,178.891,5.743,149.349
C05128=1173.923,-112.563,-40.851,178.894,5.743,149.349
C05129=1173.918,-112.313,-40.860,178.895,5.743,149.348
C05130=1173.913,-112.063,-40.869,178.898,5.744,149.348
C05131=1173.908,-111.813,-40.878,178.900,5.744,149.347
C05132=1173.902,-111.564,-40.888,178.902,5.744,149.347
C05133=1173.897,-111.314,-40.897,178.904,5.744,149.346
C05134=1173.892,-111.064,-40.906,178.906,5.745,149.345
C05135=1173.886,-110.814,-40.915,178.908,5.744,149.345
C05136=1173.881,-110.564,-40.924,178.910,5.745,149.344
C05137=1173.876,-110.315,-40.934,178.912,5.745,149.344
C05138=1173.871,-110.065,-40.943,178.915,5.745,149.343
C05139=1173.865,-109.815,-40.952,178.916,5.745,149.342
C05140=1173.860,-109.565,-40.961,178.919,5.746,149.342
C05141=1173.855,-109.315,-40.971,178.921,5.746,149.341
C05142=1173.848,-109.066,-40.980,178.923,5.746,149.341
C05143=1173.843,-108.816,-40.989,178.925,5.747,149.340
C05144=1173.838,-108.566,-40.997,178.927,5.747,149.340
C05145=1173.832,-108.317,-41.008,178.930,5.747,149.339
C05146=1173.827,-108.067,-41.017,178.931,5.747,149.338
C05147=1173.822,-107.817,-41.025,178.934,5.748,149.338
C05148=1173.816,-107.568,-41.036,178.936,5.748,149.337
C05149=1173.811,-107.318,-41.045,178.938,5.748,149.336
C05150=1173.806,-107.068,-41.053,178.940,5.748,149.336
C05151=1173.800,-106.818,-41.064,178.942,5.749,149.335
C05152=1173.796,-106.568,-41.073,178.944,5.748,149.335
C05153=1173.791,-106.318,-41.082,178.946,5.749,149.334
C05154=1173.785,-106.068,-41.092,178.949,5.749,149.334
C05155=1173.780,-105.818,-41.101,178.951,5.749,149.333
C05156=1173.775,-105.569,-41.110,178.953,5.750,149.332
C05157=1173.769,-105.319,-41.120,178.955,5.750,149.332
C05158=1173.764,-105.069,-41.129,178.957,5.751,149.331
C05159=1173.758,-104.819,-41.138,178.959,5.750,149.331
C05160=1173.753,-104.570,-41.148,178.961,5.751,149.330
C05161=1173.748,-104.320,-41.157,178.963,5.751,149.329
C05162=1173.742,-104.070,-41.167,178.966,5.751,149.329
C05163=1173.737,-103.821,-41.176,178.968,5.751,149.328
C05164=1173.731,-103.570,-41.186,178.970,5.752,149.328
C05165=1173.727,-103.321,-41.195,178.973,5.752,149.327
C05166=1173.721,-103.071,-41.204,178.974,5.752,149.327
C05167=1173.716,-102.822,-41.214,178.977,5.752,149.326
C05168=1173.711,-102.572,-41.223,178.978,5.752,149.325
C05169=1173.705,-102.300,-41.233,178.981,5.753,149.325
C05170=1173.699,-102.028,-41.244,178.983,5.754,149.324
C05171=1173.693,-101.756,-41.254,178.985,5.753,149.323
C05172=1173.687,-101.485,-41.264,178.988,5.754,149.323
C05173=1173.682,-101.235,-41.275,178.990,5.754,149.322
C05174=1173.677,-100.985,-41.284,178.992,5.754,149.322
C05175=1173.672,-100.735,-41.294,178.994,5.755,149.321
C05176=1173.666,-100.485,-41.303,178.997,5.754,149.320
C05177=1173.661,-100.236,-41.313,178.999,5.755,149.320
C05178=1173.656,-99.986,-41.322,179.001,5.756,149.319
C05179=1173.651,-99.737,-41.332,179.003,5.755,149.319
C05180=1173.645,-99.486,-41.341,179.005,5.756,149.318
C05181=1173.640,-99.237,-41.351,179.007,5.756,149.318
C05182=1173.634,-98.987,-41.360,179.010,5.757,149.317
C05183=1173.630,-98.737,-41.370,179.012,5.756,149.316
C05184=1173.624,-98.487,-41.380,179.014,5.757,149.316
C05185=1173.619,-98.238,-41.389,179.016,5.757,149.315
C05186=1173.613,-97.988,-41.400,179.018,5.757,149.315
C05187=1173.608,-97.738,-41.409,179.021,5.758,149.314
C05188=1173.603,-97.489,-41.419,179.022,5.758,149.313
C05189=1173.597,-97.239,-41.428,179.025,5.758,149.313
C05190=1173.592,-96.989,-41.438,179.027,5.758,149.312
C05191=1173.587,-96.739,-41.448,179.029,5.758,149.312
C05192=1173.582,-96.489,-41.457,179.031,5.759,149.311
C05193=1173.576,-96.240,-41.467,179.034,5.759,149.310
C05194=1173.571,-95.990,-41.476,179.036,5.760,149.310
C05195=1173.565,-95.740,-41.487,179.037,5.760,149.309
C05196=1173.560,-95.491,-41.497,179.040,5.760,149.309
C05197=1173.555,-95.241,-41.506,179.042,5.761,149.308
C05198=1173.550,-94.991,-41.516,179.044,5.760,149.307
C05199=1173.544,-94.741,-41.525,179.046,5.761,149.307
C05200=1173.539,-94.491,-41.535,179.049,5.761,149.306
C05201=1173.534,-94.242,-41.545,179.051,5.761,149.306
C05202=1173.528,-93.992,-41.554,179.053,5.762,149.305
C05203=1173.522,-93.742,-41.565,179.055,5.762,149.305
C05204=1173.518,-93.492,-41.575,179.058,5.762,149.304
C05205=1173.513,-93.243,-41.585,179.059,5.762,149.303
C05206=1173.507,-92.993,-41.594,179.062,5.763,149.303
C05207=1173.502,-92.743,-41.604,179.064,5.763,149.302
C05208=1173.496,-92.494,-41.614,179.066,5.763,149.301
C05209=1173.492,-92.243,-41.623,179.068,5.764,149.301
C05210=1173.486,-91.994,-41.634,179.070,5.763,149.300
C05211=1173.481,-91.744,-41.644,179.073,5.764,149.300
C05212=1173.475,-91.494,-41.653,179.075,5.764,149.299
C05213=1173.470,-91.245,-41.663,179.077,5.765,149.299
C05214=1173.465,-90.995,-41.673,179.080,5.765,149.298
C05215=1173.460,-90.745,-41.683,179.081,5.765,149.297
C05216=1173.454,-90.495,-41.693,179.084,5.765,149.297
C05217=1173.448,-90.246,-41.703,179.086,5.766,149.296
C05218=1173.444,-89.996,-41.713,179.088,5.766,149.296
C05219=1173.439,-89.746,-41.723,179.090,5.766,149.295
C05220=1173.433,-89.497,-41.733,179.092,5.766,149.294
C05221=1173.428,-89.247,-41.742,179.095,5.767,149.294
C05222=1173.423,-88.997,-41.753,179.097,5.767,149.293
C05223=1173.417,-88.747,-41.763,179.099,5.767,149.293
C05224=1173.412,-88.498,-41.772,179.102,5.768,149.292
C05225=1173.407,-88.248,-41.783,179.103,5.768,149.291
C05226=1173.401,-87.997,-41.793,179.106,5.768,149.291
C05227=1173.396,-87.748,-41.803,179.108,5.769,149.290
C05228=1173.391,-87.499,-41.812,179.110,5.768,149.290
C05229=1173.385,-87.249,-41.823,179.112,5.769,149.289
C05230=1173.380,-86.999,-41.833,179.115,5.770,149.288
C05231=1173.375,-86.749,-41.843,179.117,5.770,149.288
C05232=1173.370,-86.500,-41.853,179.119,5.770,149.287
C05233=1173.365,-86.249,-41.863,179.121,5.770,149.287
C05234=1173.359,-86.000,-41.873,179.124,5.770,149.286
C05235=1173.353,-85.750,-41.883,179.126,5.771,149.285
C05236=1173.349,-85.501,-41.893,179.128,5.771,149.285
C05237=1173.344,-85.251,-41.903,179.130,5.771,149.284
C05238=1173.338,-85.001,-41.914,179.133,5.772,149.284
C05239=1173.332,-84.752,-41.924,179.135,5.771,149.283
C05240=1173.328,-84.502,-41.934,179.137,5.772,149.282
C05241=1173.322,-84.252,-41.944,179.139,5.772,149.282
C05242=1173.317,-84.003,-41.954,179.141,5.773,149.281
C05243=1173.312,-83.752,-41.965,179.144,5.773,149.280
C05244=1173.306,-83.503,-41.975,179.145,5.773,149.280
C05245=1173.301,-83.253,-41.985,179.148,5.773,149.279
C05246=1173.296,-83.003,-41.995,179.150,5.774,149.279
C05247=1173.291,-82.753,-42.005,179.152,5.774,149.278
C05248=1173.285,-82.504,-42.015,179.155,5.775,149.278
C05249=1173.280,-82.253,-42.025,179.157,5.774,149.277
C05250=1173.275,-82.004,-42.035,179.159,5.775,149.276
C05251=1173.269,-81.755,-42.045,179.162,5.775,149.276
C05252=1173.264,-81.504,-42.056,179.163,5.775,149.275
C05253=1173.259,-81.255,-42.066,179.166,5.776,149.275
C05254=1173.253,-81.005,-42.076,179.168,5.777,149.274
C05255=1173.249,-80.756,-42.088,179.170,5.776,149.273
C05256=1173.243,-80.506,-42.098,179.173,5.777,149.273
C05257=1173.238,-80.257,-42.107,179.175,5.777,149.272
C05258=1173.233,-80.007,-42.118,179.177,5.777,149.271
C05259=1173.228,-79.757,-42.128,179.179,5.778,149.271
C05260=1173.222,-79.507,-42.138,179.182,5.778,149.270
C05261=1173.217,-79.257,-42.149,179.183,5.778,149.270
C05262=1173.211,-79.008,-42.159,179.186,5.779,149.269
C05263=1173.206,-78.757,-42.170,179.188,5.779,149.269
C05264=1173.201,-78.508,-42.180,179.190,5.779,149.268
C05265=1173.195,-78.258,-42.190,179.193,5.780,149.267
C05266=1173.190,-78.008,-42.201,179.195,5.779,149.267
C05267=1173.185,-77.759,-42.210,179.197,5.780,149.266
C05268=1173.181,-77.509,-42.222,179.200,5.781,149.265
C05269=1173.175,-77.260,-42.232,179.202,5.780,149.265
C05270=1173.169,-77.010,-42.242,179.204,5.781,149.264
C05271=1173.164,-76.760,-42.253,179.206,5.781,149.264
C05272=1173.159,-76.510,-42.263,179.208,5.781,149.263
C05273=1173.153,-76.239,-42.274,179.211,5.782,149.262
C05274=1173.147,-75.969,-42.286,179.213,5.782,149.262
C05275=1173.141,-75.697,-42.297,179.216,5.783,149.261
C05276=1173.136,-75.426,-42.308,179.218,5.783,149.260
C05277=1173.131,-75.176,-42.318,179.220,5.783,149.260
C05278=1173.126,-74.926,-42.329,179.223,5.784,149.259
C05279=1173.120,-74.677,-42.340,179.225,5.784,149.259
C05280=1173.115,-74.427,-42.350,179.227,5.784,149.258
C05281=1173.110,-74.177,-42.361,179.229,5.785,149.257
C05282=1173.104,-73.928,-42.371,179.232,5.785,149.257
C05283=1173.100,-73.678,-42.382,179.234,5.785,149.256
C05284=1173.094,-73.429,-42.392,179.236,5.785,149.256
C05285=1173.088,-73.178,-42.404,179.239,5.786,149.255
C05286=1173.083,-72.929,-42.414,179.241,5.786,149.254
C05287=1173.078,-72.678,-42.424,179.243,5.787,149.254
C05288=1173.072,-72.429,-42.435,179.246,5.787,149.253
C05289=1173.067,-72.179,-42.446,179.247,5.787,149.253
C05290=1173.062,-71.930,-42.456,179.250,5.787,149.252
C05291=1173.057,-71.680,-42.467,179.252,5.788,149.251
C05292=1173.051,-71.430,-42.478,179.254,5.788,149.251
C05293=1173.046,-71.180,-42.488,179.257,5.788,149.250
C05294=1173.041,-70.931,-42.498,179.259,5.789,149.250
C05295=1173.036,-70.681,-42.510,179.262,5.789,149.249
C05296=1173.031,-70.431,-42.520,179.263,5.789,149.248
C05297=1173.026,-70.181,-42.530,179.266,5.790,149.248
C05298=1173.020,-69.932,-42.541,179.269,5.790,149.247
C05299=1173.015,-69.682,-42.552,179.270,5.790,149.246
C05300=1173.010,-69.433,-42.562,179.273,5.791,149.246
C05301=1173.004,-69.183,-42.574,179.275,5.791,149.245
C05302=1172.999,-68.933,-42.584,179.277,5.791,149.245
C05303=1172.994,-68.683,-42.595,179.279,5.792,149.244
C05304=1172.988,-68.434,-42.606,179.282,5.792,149.243
C05305=1172.983,-68.184,-42.616,179.284,5.792,149.243
C05306=1172.978,-67.935,-42.627,179.286,5.793,149.242
C05307=1172.973,-67.684,-42.638,179.289,5.793,149.242
C05308=1172.967,-67.435,-42.648,179.291,5.794,149.241
C05309=1172.962,-67.185,-42.660,179.293,5.793,149.240
C05310=1172.956,-66.935,-42.670,179.295,5.794,149.240
C05311=1172.952,-66.686,-42.681,179.298,5.795,149.239
C05312=1172.946,-66.436,-42.692,179.300,5.794,149.238
C05313=1172.941,-66.187,-42.703,179.302,5.795,149.238
C05314=1172.936,-65.936,-42.713,179.305,5.795,149.237
C05315=1172.931,-65.687,-42.724,179.306,5.795,149.237
C05316=1172.925,-65.437,-42.736,179.309,5.796,149.236
C05317=1172.920,-65.187,-42.746,179.311,5.797,149.236
C05318=1172.915,-64.938,-42.757,179.314,5.797,149.235
C05319=1172.909,-64.688,-42.767,179.316,5.797,149.234
C05320=1172.905,-64.439,-42.779,179.318,5.797,149.234
C05321=1172.899,-64.188,-42.790,179.321,5.798,149.233
C05322=1172.894,-63.939,-42.801,179.323,5.798,149.233
C05323=1172.889,-63.689,-42.811,179.325,5.798,149.232
C05324=1172.883,-63.440,-42.822,179.327,5.799,149.231
C05325=1172.878,-63.190,-42.833,179.330,5.799,149.231
C05326=1172.873,-62.940,-42.845,179.332,5.799,149.230
C05327=1172.868,-62.691,-42.855,179.334,5.800,149.229
C05328=1172.863,-62.441,-42.866,179.337,5.800,149.229
C05329=1172.857,-62.192,-42.877,179.339,5.801,149.228
C05330=1172.852,-61.941,-42.888,179.341,5.801,149.228
C05331=1172.847,-61.691,-42.899,179.344,5.801,149.227
C05332=1172.841,-61.442,-42.910,179.346,5.802,149.226
C05333=1172.837,-61.192,-42.921,179.348,5.801,149.226
C05334=1172.831,-60.942,-42.933,179.350,5.802,149.225
C05335=1172.826,-60.693,-42.943,179.353,5.803,149.224
C05336=1172.821,-60.443,-42.954,179.355,5.803,149.224
C05337=1172.815,-60.194,-42.965,179.357,5.803,149.223
C05338=1172.810,-59.944,-42.976,179.360,5.804,149.223
C05339=1172.805,-59.694,-42.988,179.362,5.804,149.222
C05340=1172.800,-59.445,-42.998,179.365,5.805,149.221
C05341=1172.794,-59.195,-43.010,179.366,5.805,149.221
C05342=1172.790,-58.945,-43.021,179.369,5.805,149.220
C05343=1172.784,-58.695,-43.031,179.372,5.806,149.220
C05344=1172.779,-58.446,-43.043,179.373,5.806,149.219
C05345=1172.774,-58.196,-43.054,179.376,5.806,149.218
C05346=1172.768,-57.946,-43.065,179.378,5.807,149.218
C05347=1172.764,-57.697,-43.076,179.381,5.807,149.217
C05348=1172.758,-57.447,-43.088,179.383,5.807,149.216
C05349=1172.753,-57.197,-43.098,179.385,5.808,149.216
C05350=1172.748,-56.948,-43.109,179.388,5.808,149.215
C05351=1172.742,-56.698,-43.121,179.390,5.809,149.215
C05352=1172.737,-56.447,-43.132,179.392,5.808,149.214
C05353=1172.732,-56.199,-43.143,179.394,5.809,149.214
C05354=1172.727,-55.949,-43.155,179.397,5.810,149.213
C05355=1172.722,-55.699,-43.166,179.400,5.810,149.212
C05356=1172.716,-55.449,-43.177,179.401,5.810,149.212
C05357=1172.711,-55.199,-43.188,179.404,5.811,149.211
C05358=1172.706,-54.950,-43.199,179.406,5.811,149.211
C05359=1172.701,-54.700,-43.211,179.409,5.812,149.210
C05360=1172.696,-54.451,-43.222,179.411,5.811,149.209
C05361=1172.691,-54.201,-43.233,179.413,5.812,149.209
C05362=1172.685,-53.951,-43.245,179.416,5.813,149.208
C05363=1172.680,-53.701,-43.256,179.418,5.813,149.207
C05364=1172.674,-53.452,-43.267,179.420,5.814,149.207
C05365=1172.670,-53.202,-43.279,179.423,5.813,149.206
C05366=1172.664,-52.952,-43.290,179.425,5.814,149.206
C05367=1172.659,-52.702,-43.301,179.427,5.815,149.205
C05368=1172.654,-52.453,-43.312,179.430,5.815,149.204
C05369=1172.649,-52.203,-43.324,179.432,5.815,149.204
C05370=1172.644,-51.954,-43.335,179.434,5.815,149.203
C05371=1172.638,-51.704,-43.347,179.437,5.816,149.203
C05372=1172.633,-51.455,-43.358,179.439,5.817,149.202
C05373=1172.627,-51.204,-43.369,179.441,5.817,149.201
C05374=1172.623,-50.955,-43.381,179.443,5.817,149.201
C05375=1172.617,-50.705,-43.392,179.446,5.818,149.200
C05376=1172.612,-50.456,-43.403,179.448,5.818,149.199
C05377=1172.607,-50.185,-43.416,179.451,5.819,149.199
C05378=1172.601,-49.914,-43.429,179.454,5.819,149.198
C05379=1172.595,-49.644,-43.440,179.456,5.820,149.197
C05380=1172.590,-49.374,-43.453,179.458,5.819,149.197
C05381=1172.585,-49.124,-43.465,179.461,5.820,149.196
C05382=1172.579,-48.874,-43.477,179.463,5.820,149.195
C05383=1172.574,-48.625,-43.487,179.465,5.821,149.195
C05384=1172.569,-48.375,-43.499,179.468,5.822,149.194
C05385=1172.563,-48.125,-43.511,179.470,5.821,149.194
C05386=1172.559,-47.876,-43.523,179.472,5.822,149.193
C05387=1172.553,-47.626,-43.534,179.475,5.823,149.192
C05388=1172.548,-47.377,-43.545,179.477,5.823,149.192
C05389=1172.542,-47.127,-43.557,179.480,5.824,149.191
C05390=1172.538,-46.877,-43.569,179.482,5.823,149.191
C05391=1172.532,-46.627,-43.580,179.484,5.824,149.190
C05392=1172.527,-46.377,-43.592,179.487,5.825,149.189
C05393=1172.522,-46.128,-43.604,179.489,5.825,149.189
C05394=1172.516,-45.879,-43.615,179.491,5.825,149.188
C05395=1172.511,-45.629,-43.626,179.494,5.825,149.187
C05396=1172.506,-45.379,-43.638,179.496,5.826,149.187
C05397=1172.501,-45.129,-43.650,179.499,5.827,149.186
C05398=1172.496,-44.880,-43.661,179.501,5.827,149.186
C05399=1172.491,-44.630,-43.673,179.503,5.827,149.185
C05400=1172.486,-44.380,-43.685,179.505,5.828,149.184
C05401=1172.480,-44.131,-43.696,179.508,5.828,149.184
C05402=1172.474,-43.881,-43.708,179.510,5.829,149.183
C05403=1172.470,-43.631,-43.719,179.513,5.829,149.183
C05404=1172.465,-43.382,-43.732,179.515,5.830,149.182
C05405=1172.460,-43.132,-43.743,179.517,5.830,149.181
C05406=1172.454,-42.882,-43.755,179.520,5.830,149.181
C05407=1172.449,-42.632,-43.767,179.522,5.831,149.180
C05408=1172.444,-42.383,-43.778,179.525,5.831,149.179
C05409=1172.439,-42.133,-43.790,179.527,5.832,149.179
C05410=1172.433,-41.884,-43.802,179.529,5.832,149.178
C05411=1172.428,-41.635,-43.814,179.532,5.832,149.178
C05412=1172.423,-41.385,-43.826,179.534,5.833,149.177
C05413=1172.418,-41.135,-43.837,179.537,5.833,149.176
C05414=1172.413,-40.885,-43.849,179.539,5.834,149.176
C05415=1172.407,-40.635,-43.861,179.541,5.834,149.175
C05416=1172.402,-40.386,-43.873,179.543,5.834,149.175
C05417=1172.397,-40.136,-43.885,179.546,5.835,149.174
C05418=1172.392,-39.886,-43.896,179.548,5.836,149.173
C05419=1172.387,-39.636,-43.908,179.551,5.836,149.173
C05420=1172.381,-39.386,-43.920,179.553,5.837,149.172
C05421=1172.376,-39.137,-43.933,179.555,5.836,149.172
C05422=1172.372,-38.887,-43.944,179.557,5.837,149.171
C05423=1172.366,-38.638,-43.956,179.560,5.838,149.170
C05424=1172.360,-38.388,-43.967,179.563,5.838,149.170
C05425=1172.355,-38.139,-43.980,179.565,5.839,149.169
C05426=1172.350,-37.889,-43.991,179.568,5.839,149.168
C05427=1172.345,-37.639,-44.003,179.570,5.839,149.168
C05428=1172.340,-37.390,-44.016,179.572,5.840,149.167
C05429=1172.334,-37.140,-44.028,179.574,5.840,149.167
C05430=1172.330,-36.890,-44.039,179.577,5.841,149.166
C05431=1172.324,-36.641,-44.051,179.579,5.841,149.165
C05432=1172.319,-36.391,-44.064,179.582,5.842,149.165
C05433=1172.314,-36.141,-44.075,179.584,5.842,149.164
C05434=1172.308,-35.891,-44.087,179.586,5.842,149.164
C05435=1172.304,-35.642,-44.099,179.589,5.843,149.163
C05436=1172.298,-35.392,-44.111,179.591,5.844,149.162
C05437=1172.293,-35.143,-44.124,179.594,5.844,149.162
C05438=1172.288,-34.893,-44.136,179.596,5.845,149.161
C05439=1172.282,-34.643,-44.148,179.599,5.845,149.161
C05440=1172.277,-34.394,-44.160,179.601,5.845,149.160
C05441=1172.273,-34.144,-44.171,179.603,5.846,149.159
C05442=1172.267,-33.894,-44.183,179.605,5.846,149.159
C05443=1172.262,-33.645,-44.196,179.608,5.847,149.158
C05444=1172.257,-33.395,-44.208,179.610,5.847,149.157
C05445=1172.251,-33.146,-44.220,179.613,5.848,149.157
C05446=1172.246,-32.896,-44.232,179.615,5.849,149.156
C05447=1172.241,-32.647,-44.245,179.617,5.848,149.156
C05448=1172.236,-32.397,-44.256,179.620,5.849,149.155
C05449=1172.231,-32.148,-44.269,179.622,5.850,149.154
C05450=1172.226,-31.898,-44.281,179.625,5.850,149.154
C05451=1172.220,-31.648,-44.293,179.627,5.850,149.153
C05452=1172.216,-31.398,-44.306,179.630,5.851,149.153
C05453=1172.210,-31.148,-44.317,179.632,5.852,149.152
C05454=1172.205,-30.898,-44.330,179.634,5.852,149.151
C05455=1172.200,-30.648,-44.342,179.637,5.852,149.151
C05456=1172.195,-30.399,-44.354,179.639,5.853,149.150
C05457=1172.189,-30.149,-44.366,179.641,5.853,149.150
C05458=1172.184,-29.900,-44.379,179.644,5.854,149.149
C05459=1172.180,-29.651,-44.391,179.647,5.854,149.148
C05460=1172.174,-29.401,-44.403,179.649,5.855,149.148
C05461=1172.169,-29.152,-44.415,179.652,5.855,149.147
C05462=1172.164,-28.902,-44.427,179.653,5.855,149.146
C05463=1172.159,-28.652,-44.440,179.656,5.856,149.146
C05464=1172.154,-28.402,-44.452,179.658,5.856,149.145
C05465=1172.149,-28.152,-44.465,179.661,5.857,149.145
C05466=1172.143,-27.903,-44.477,179.663,5.858,149.144
C05467=1172.138,-27.653,-44.489,179.666,5.858,149.143
C05468=1172.133,-27.404,-44.502,179.668,5.859,149.143
C05469=1172.128,-27.154,-44.514,179.671,5.859,149.142
C05470=1172.122,-26.905,-44.526,179.673,5.860,149.142
C05471=1172.117,-26.655,-44.539,179.675,5.860,149.141
C05472=1172.112,-26.405,-44.551,179.678,5.860,149.140
C05473=1172.107,-26.155,-44.564,179.680,5.861,149.140
C05474=1172.102,-25.906,-44.576,179.683,5.861,149.139
C05475=1172.097,-25.656,-44.588,179.685,5.862,149.138
C05476=1172.092,-25.407,-44.601,179.687,5.863,149.138
C05477=1172.087,-25.157,-44.614,179.690,5.863,149.137
C05478=1172.081,-24.908,-44.625,179.693,5.864,149.136
C05479=1172.077,-24.657,-44.638,179.695,5.864,149.136
C05480=1172.071,-24.408,-44.651,179.698,5.865,149.135
C05481=1172.065,-24.138,-44.664,179.700,5.865,149.135
C05482=1172.060,-23.868,-44.678,179.703,5.866,149.134
C05483=1172.055,-23.599,-44.692,179.705,5.867,149.133
C05484=1172.048,-23.329,-44.705,179.708,5.867,149.133
C05485=1172.044,-23.079,-44.718,179.710,5.867,149.132
C05486=1172.038,-22.829,-44.730,179.713,5.868,149.132
C05487=1172.033,-22.580,-44.742,179.715,5.868,149.131
C05488=1172.028,-22.330,-44.755,179.717,5.868,149.130
C05489=1172.023,-22.081,-44.767,179.719,5.869,149.130
C05490=1172.018,-21.832,-44.780,179.722,5.870,149.129
C05491=1172.012,-21.581,-44.794,179.725,5.870,149.128
C05492=1172.007,-21.331,-44.805,179.727,5.871,149.128
C05493=1172.002,-21.082,-44.818,179.730,5.871,149.127
C05494=1171.997,-20.833,-44.831,179.732,5.872,149.126
C05495=1171.992,-20.583,-44.844,179.734,5.873,149.126
C05496=1171.987,-20.333,-44.856,179.737,5.873,149.125
